C07272=1095.024,419.348,-100.142,178.825,23.629,153.449
C07273=1095.018,419.101,-100.102,178.823,23.620,153.447
C07274=1095.011,418.855,-100.061,178.820,23.611,153.445
C07275=1095.006,418.608,-100.020,178.817,23.601,153.443
C07276=1095.000,418.362,-99.979,178.814,23.592,153.441
C07277=1094.993,418.116,-99.938,178.811,23.583,153.439
C07278=1094.987,417.868,-99.897,178.808,23.573,153.437
C07279=1094.982,417.653,-99.862,178.806,23.565,153.436
C07280=1094.976,417.437,-99.827,178.804,23.558,153.434
C07281=1094.972,417.222,-99.791,178.802,23.550,153.433
C07282=1094.966,417.006,-99.756,178.799,23.542,153.431
C07283=1094.960,416.791,-99.720,178.797,23.534,153.429
C07284=1094.956,416.575,-99.685,178.794,23.526,153.428
C07285=1094.950,416.359,-99.649,178.792,23.518,153.426
C07286=1094.945,416.144,-99.613,178.789,23.510,153.424
C07287=1094.938,415.897,-99.573,178.786,23.501,153.423
C07288=1094.933,415.650,-99.533,178.783,23.492,153.421
C07289=1094.926,415.404,-99.492,178.780,23.483,153.419
C07290=1094.920,415.157,-99.452,178.778,23.475,153.417
C07291=1094.914,414.910,-99.411,178.776,23.466,153.415
C07292=1094.908,414.664,-99.371,178.772,23.457,153.414
C07293=1094.902,414.417,-99.331,178.770,23.448,153.412
C07294=1094.896,414.170,-99.290,178.767,23.439,153.410
C07295=1094.890,413.923,-99.251,178.764,23.431,153.408
C07296=1094.883,413.677,-99.211,178.762,23.422,153.407
C07297=1094.877,413.430,-99.171,178.758,23.414,153.405
C07298=1094.871,413.184,-99.130,178.756,23.405,153.403
C07299=1094.865,412.937,-99.090,178.753,23.396,153.401
C07300=1094.859,412.690,-99.050,178.750,23.387,153.400
C07301=1094.853,412.443,-99.010,178.747,23.379,153.398
C07302=1094.847,412.197,-98.970,178.744,23.371,153.396
C07303=1094.841,411.951,-98.930,178.741,23.362,153.395
C07304=1094.835,411.704,-98.890,178.738,23.353,153.393
C07305=1094.829,411.457,-98.850,178.736,23.345,153.391
C07306=1094.823,411.210,-98.809,178.733,23.337,153.390
C07307=1094.816,410.955,-98.768,178.730,23.328,153.388
C07308=1094.810,410.698,-98.727,178.727,23.319,153.386
C07309=1094.804,410.442,-98.686,178.724,23.311,153.384
C07310=1094.798,410.186,-98.644,178.721,23.302,153.383
C07311=1094.791,409.939,-98.604,178.719,23.294,153.381
C07312=1094.785,409.692,-98.565,178.716,23.286,153.379
C07313=1094.780,409.446,-98.524,178.713,23.277,153.378
C07314=1094.774,409.199,-98.485,178.711,23.269,153.376
C07315=1094.768,408.952,-98.445,178.708,23.261,153.374
C07316=1094.762,408.705,-98.405,178.705,23.253,153.373
C07317=1094.755,408.459,-98.365,178.702,23.245,153.371
C07318=1094.750,408.212,-98.326,178.699,23.237,153.370
C07319=1094.744,407.965,-98.287,178.696,23.228,153.368
C07320=1094.738,407.718,-98.246,178.694,23.220,153.366
C07321=1094.732,407.471,-98.207,178.691,23.212,153.365
C07322=1094.727,407.225,-98.167,178.688,23.205,153.363
C07323=1094.720,406.978,-98.127,178.685,23.196,153.362
C07324=1094.714,406.731,-98.088,178.682,23.188,153.360
C07325=1094.708,406.484,-98.048,178.680,23.180,153.359
C07326=1094.703,406.237,-98.009,178.677,23.172,153.357
C07327=1094.695,405.991,-97.970,178.674,23.164,153.356
C07328=1094.689,405.744,-97.930,178.671,23.156,153.354
C07329=1094.683,405.497,-97.891,178.669,23.149,153.353
C07330=1094.678,405.250,-97.852,178.666,23.141,153.351
C07331=1094.672,405.003,-97.812,178.663,23.133,153.349
C07332=1094.666,404.756,-97.773,178.660,23.126,153.348
C07333=1094.660,404.510,-97.734,178.657,23.118,153.347
C07334=1094.654,404.263,-97.695,178.655,23.110,153.345
C07335=1094.648,404.015,-97.655,178.651,23.102,153.344
C07336=1094.642,403.769,-97.617,178.649,23.095,153.342
C07337=1094.636,403.522,-97.577,178.646,23.087,153.341
C07338=1094.630,403.275,-97.538,178.643,23.080,153.339
C07339=1094.624,403.029,-97.499,178.640,23.072,153.338
C07340=1094.617,402.782,-97.460,178.638,23.064,153.336
C07341=1094.611,402.535,-97.420,178.635,23.057,153.335
C07342=1094.606,402.288,-97.381,178.632,23.049,153.333
C07343=1094.600,402.041,-97.342,178.630,23.042,153.332
C07344=1094.593,401.794,-97.303,178.626,23.034,153.331
C07345=1094.588,401.548,-97.264,178.624,23.027,153.329
C07346=1094.581,401.301,-97.225,178.620,23.019,153.328
C07347=1094.576,401.054,-97.186,178.618,23.012,153.326
C07348=1094.569,400.807,-97.147,178.615,23.005,153.325
C07349=1094.564,400.560,-97.108,178.612,22.997,153.324
C07350=1094.558,400.313,-97.069,178.610,22.990,153.322
C07351=1094.551,400.066,-97.031,178.607,22.982,153.321
C07352=1094.546,399.819,-96.992,178.604,22.975,153.319
C07353=1094.540,399.572,-96.952,178.601,22.968,153.318
C07354=1094.534,399.326,-96.915,178.598,22.961,153.317
C07355=1094.528,399.078,-96.875,178.596,22.954,153.315
C07356=1094.522,398.832,-96.837,178.592,22.946,153.314
C07357=1094.516,398.584,-96.798,178.590,22.939,153.313
C07358=1094.510,398.338,-96.759,178.587,22.932,153.311
C07359=1094.504,398.118,-96.725,178.585,22.926,153.310
C07360=1094.499,397.898,-96.691,178.582,22.919,153.309
C07361=1094.493,397.677,-96.656,178.579,22.913,153.308
C07362=1094.489,397.458,-96.621,178.577,22.907,153.306
C07363=1094.483,397.237,-96.586,178.575,22.900,153.305
C07364=1094.478,397.017,-96.552,178.572,22.894,153.304
C07365=1094.473,396.798,-96.518,178.569,22.888,153.303
C07366=1094.468,396.577,-96.484,178.567,22.882,153.302
C07367=1094.461,396.331,-96.445,178.564,22.874,153.301
C07368=1094.455,396.083,-96.407,178.561,22.868,153.299
C07369=1094.450,395.836,-96.369,178.559,22.861,153.298
C07370=1094.443,395.590,-96.330,178.556,22.854,153.297
C07371=1094.438,395.343,-96.292,178.553,22.847,153.295
C07372=1094.432,395.096,-96.254,178.550,22.840,153.294
C07373=1094.426,394.849,-96.214,178.548,22.833,153.293
C07374=1094.420,394.602,-96.177,178.544,22.826,153.292
C07375=1094.414,394.355,-96.139,178.541,22.819,153.290
C07376=1094.408,394.108,-96.099,178.539,22.813,153.289
C07377=1094.402,393.861,-96.062,178.536,22.806,153.288
C07378=1094.396,393.615,-96.024,178.533,22.799,153.287
C07379=1094.390,393.367,-95.985,178.530,22.792,153.285
C07380=1094.384,393.121,-95.947,178.527,22.786,153.284
C07381=1094.378,392.874,-95.909,178.525,22.779,153.283
C07382=1094.372,392.626,-95.871,178.521,22.772,153.282
C07383=1094.366,392.379,-95.833,178.519,22.765,153.281
C07384=1094.361,392.133,-95.795,178.516,22.759,153.279
C07385=1094.354,391.885,-95.757,178.513,22.752,153.278
C07386=1094.348,391.638,-95.719,178.511,22.746,153.277
C07387=1094.342,391.392,-95.681,178.507,22.739,153.276
C07388=1094.336,391.144,-95.643,178.504,22.732,153.275
C07389=1094.330,390.898,-95.605,178.502,22.726,153.274
C07390=1094.324,390.651,-95.566,178.499,22.720,153.272
C07391=1094.318,390.403,-95.529,178.496,22.713,153.271
C07392=1094.312,390.156,-95.491,178.493,22.706,153.270
C07393=1094.306,389.910,-95.453,178.490,22.700,153.269
C07394=1094.300,389.663,-95.416,178.487,22.694,153.268
C07395=1094.295,389.416,-95.378,178.485,22.687,153.267
C07396=1094.288,389.169,-95.340,178.482,22.681,153.266
C07397=1094.282,388.922,-95.302,178.478,22.674,153.265
C07398=1094.276,388.675,-95.264,178.475,22.668,153.263
C07399=1094.270,388.428,-95.226,178.473,22.662,153.262
C07400=1094.264,388.182,-95.189,178.470,22.655,153.261
C07401=1094.258,387.934,-95.151,178.467,22.649,153.260
C07402=1094.252,387.687,-95.113,178.464,22.643,153.259
C07403=1094.246,387.440,-95.076,178.461,22.636,153.258
C07404=1094.240,387.193,-95.038,178.458,22.630,153.257
C07405=1094.235,386.947,-95.000,178.455,22.624,153.256
C07406=1094.229,386.699,-94.963,178.452,22.617,153.254
C07407=1094.223,386.453,-94.925,178.450,22.611,153.253
C07408=1094.217,386.205,-94.887,178.447,22.605,153.252
C07409=1094.211,385.958,-94.850,178.444,22.599,153.251
C07410=1094.205,385.711,-94.812,178.441,22.593,153.250
C07411=1094.199,385.464,-94.775,178.438,22.586,153.249
C07412=1094.194,385.217,-94.738,178.435,22.580,153.248
C07413=1094.188,384.970,-94.700,178.432,22.574,153.247
C07414=1094.182,384.723,-94.663,178.429,22.568,153.246
C07415=1094.177,384.509,-94.630,178.427,22.563,153.245
C07416=1094.172,384.296,-94.598,178.424,22.557,153.244
C07417=1094.166,384.082,-94.566,178.422,22.552,153.243
C07418=1094.161,383.869,-94.534,178.420,22.547,153.242
C07419=1094.156,383.655,-94.502,178.417,22.542,153.242
C07420=1094.151,383.441,-94.469,178.415,22.536,153.240
C07421=1094.146,383.228,-94.437,178.411,22.531,153.240
C07422=1094.142,383.014,-94.405,178.409,22.525,153.239
C07423=1094.136,382.767,-94.367,178.406,22.519,153.238
C07424=1094.130,382.520,-94.330,178.404,22.514,153.237
C07425=1094.124,382.273,-94.294,178.401,22.508,153.236
C07426=1094.118,382.026,-94.256,178.398,22.502,153.235
C07427=1094.112,381.778,-94.218,178.395,22.496,153.234
C07428=1094.105,381.531,-94.182,178.392,22.490,153.233
C07429=1094.099,381.284,-94.144,178.389,22.485,153.232
C07430=1094.094,381.037,-94.107,178.386,22.479,153.231
C07431=1094.087,380.790,-94.071,178.383,22.473,153.230
C07432=1094.081,380.543,-94.033,178.380,22.467,153.229
C07433=1094.076,380.296,-93.996,178.377,22.461,153.228
C07434=1094.070,380.049,-93.959,178.374,22.455,153.227
C07435=1094.064,379.801,-93.922,178.371,22.450,153.226
C07436=1094.058,379.554,-93.885,178.369,22.444,153.225
C07437=1094.052,379.308,-93.849,178.366,22.438,153.224
C07438=1094.047,379.061,-93.812,178.363,22.432,153.223
C07439=1094.040,378.814,-93.775,178.360,22.427,153.222
C07440=1094.035,378.567,-93.738,178.357,22.421,153.221
C07441=1094.029,378.319,-93.701,178.354,22.415,153.220
C07442=1094.023,378.072,-93.665,178.351,22.409,153.220
C07443=1094.017,377.825,-93.628,178.348,22.403,153.218
C07444=1094.011,377.578,-93.591,178.345,22.398,153.218
C07445=1094.005,377.330,-93.554,178.342,22.392,153.217
C07446=1093.999,377.083,-93.518,178.339,22.386,153.216
C07447=1093.993,376.836,-93.481,178.336,22.381,153.215
C07448=1093.988,376.589,-93.444,178.333,22.375,153.214
C07449=1093.982,376.342,-93.407,178.330,22.370,153.213
C07450=1093.976,376.095,-93.370,178.327,22.364,153.212
C07451=1093.970,375.848,-93.334,178.324,22.358,153.211
C07452=1093.965,375.600,-93.297,178.321,22.353,153.210
C07453=1093.958,375.353,-93.261,178.318,22.347,153.209
C07454=1093.953,375.105,-93.224,178.315,22.342,153.209
C07455=1093.947,374.859,-93.188,178.312,22.336,153.208
C07456=1093.942,374.612,-93.151,178.309,22.331,153.207
C07457=1093.935,374.365,-93.115,178.307,22.325,153.206
C07458=1093.930,374.117,-93.078,178.304,22.320,153.205
C07459=1093.924,373.870,-93.042,178.301,22.314,153.204
C07460=1093.917,373.623,-93.005,178.298,22.309,153.203
C07461=1093.912,373.376,-92.969,178.295,22.304,153.203
C07462=1093.906,373.129,-92.932,178.292,22.298,153.202
C07463=1093.900,372.881,-92.897,178.289,22.293,153.201
C07464=1093.894,372.634,-92.860,178.285,22.287,153.200
C07465=1093.888,372.387,-92.823,178.282,22.282,153.199
C07466=1093.883,372.140,-92.788,178.280,22.277,153.198
C07467=1093.876,371.893,-92.751,178.277,22.272,153.198
C07468=1093.871,371.645,-92.715,178.274,22.266,153.197
C07469=1093.865,371.398,-92.678,178.271,22.261,153.196
C07470=1093.858,371.151,-92.642,178.268,22.255,153.195
C07471=1093.849,370.751,-92.584,178.263,22.247,153.194
C07472=1093.840,370.351,-92.526,178.258,22.238,153.192
C07473=1093.830,369.951,-92.467,178.254,22.230,153.191
C07474=1093.821,369.552,-92.409,178.249,22.222,153.190
C07475=1093.815,369.304,-92.373,178.246,22.217,153.189
C07476=1093.808,369.057,-92.337,178.243,22.211,153.188
C07477=1093.804,368.810,-92.301,178.240,22.206,153.187
C07478=1093.798,368.562,-92.265,178.236,22.201,153.187
C07479=1093.791,368.315,-92.229,178.234,22.196,153.186
C07480=1093.785,368.067,-92.193,178.231,22.190,153.185
C07481=1093.780,367.820,-92.157,178.228,22.185,153.184
C07482=1093.774,367.573,-92.120,178.225,22.180,153.184
C07483=1093.769,367.326,-92.085,178.222,22.175,153.183
C07484=1093.763,367.078,-92.049,178.218,22.170,153.182
C07485=1093.757,366.831,-92.014,178.216,22.165,153.181
C07486=1093.751,366.584,-91.977,178.213,22.160,153.180
C07487=1093.745,366.337,-91.942,178.210,22.155,153.180
C07488=1093.739,366.089,-91.906,178.207,22.150,153.179
C07489=1093.734,365.842,-91.871,178.204,22.144,153.178
C07490=1093.728,365.594,-91.835,178.201,22.140,153.177
C07491=1093.722,365.347,-91.799,178.198,22.135,153.177
C07492=1093.716,365.100,-91.763,178.195,22.130,153.176
C07493=1093.710,364.853,-91.727,178.192,22.125,153.175
C07494=1093.704,364.606,-91.692,178.189,22.120,153.175
C07495=1093.698,364.358,-91.656,178.186,22.115,153.174
C07496=1093.692,364.110,-91.621,178.183,22.110,153.173
C07497=1093.687,363.863,-91.585,178.180,22.105,153.172
C07498=1093.681,363.616,-91.549,178.177,22.101,153.172
C07499=1093.675,363.369,-91.514,178.174,22.095,153.171
C07500=1093.669,363.121,-91.478,178.171,22.090,153.170
C07501=1093.663,362.873,-91.443,178.168,22.085,153.170
C07502=1093.658,362.626,-91.407,178.165,22.081,153.169
C07503=1093.652,362.379,-91.372,178.162,22.076,153.168
C07504=1093.647,362.132,-91.336,178.159,22.071,153.168
C07505=1093.640,361.884,-91.301,178.156,22.066,153.167
C07506=1093.635,361.637,-91.266,178.153,22.061,153.166
C07507=1093.629,361.389,-91.231,178.150,22.057,153.166
C07508=1093.623,361.141,-91.195,178.147,22.052,153.165
C07509=1093.617,360.894,-91.160,178.143,22.047,153.164
C07510=1093.611,360.647,-91.124,178.141,22.042,153.163
C07511=1093.605,360.400,-91.089,178.138,22.038,153.163
C07512=1093.599,360.152,-91.054,178.135,22.032,153.162
C07513=1093.594,359.905,-91.019,178.132,22.028,153.161
C07514=1093.588,359.657,-90.983,178.129,22.024,153.161
C07515=1093.583,359.409,-90.948,178.126,22.018,153.160
C07516=1093.576,359.162,-90.913,178.122,22.014,153.160
C07517=1093.570,358.915,-90.878,178.120,22.009,153.159
C07518=1093.564,358.667,-90.842,178.117,22.004,153.158
C07519=1093.559,358.420,-90.808,178.113,22.000,153.158
C07520=1093.553,358.172,-90.772,178.111,21.995,153.157
C07521=1093.547,357.925,-90.738,178.107,21.991,153.156
C07522=1093.541,357.678,-90.703,178.104,21.986,153.156
C07523=1093.532,357.293,-90.649,178.100,21.979,153.155
C07524=1093.523,356.908,-90.593,178.095,21.972,153.154
C07525=1093.514,356.524,-90.539,178.091,21.965,153.153
C07526=1093.505,356.139,-90.485,178.085,21.957,153.152
C07527=1093.499,355.892,-90.450,178.083,21.953,153.151
C07528=1093.493,355.644,-90.415,178.080,21.948,153.151
C07529=1093.488,355.397,-90.380,178.076,21.943,153.150
C07530=1093.482,355.150,-90.346,178.074,21.939,153.149
C07531=1093.476,354.902,-90.310,178.070,21.934,153.149
C07532=1093.470,354.655,-90.276,178.067,21.930,153.148
C07533=1093.464,354.406,-90.241,178.065,21.926,153.147
C07534=1093.459,354.160,-90.206,178.061,21.921,153.147
C07535=1093.453,353.912,-90.172,178.059,21.917,153.146
C07536=1093.447,353.664,-90.137,178.055,21.912,153.146
C07537=1093.441,353.417,-90.102,178.052,21.908,153.145
C07538=1093.436,353.170,-90.067,178.049,21.903,153.145
C07539=1093.430,352.922,-90.033,178.046,21.899,153.144
C07540=1093.425,352.674,-89.998,178.043,21.894,153.143
C07541=1093.418,352.427,-89.963,178.040,21.890,153.143
C07542=1093.412,352.179,-89.929,178.037,21.886,153.142
C07543=1093.407,351.932,-89.894,178.034,21.881,153.142
C07544=1093.400,351.684,-89.860,178.031,21.877,153.141
C07545=1093.395,351.436,-89.825,178.027,21.872,153.141
C07546=1093.389,351.190,-89.791,178.025,21.868,153.140
C07547=1093.383,350.942,-89.756,178.021,21.864,153.140
C07548=1093.377,350.694,-89.721,178.019,21.860,153.139
C07549=1093.372,350.447,-89.687,178.016,21.855,153.138
C07550=1093.367,350.199,-89.653,178.012,21.851,153.138
C07551=1093.360,349.951,-89.618,178.010,21.846,153.137
C07552=1093.354,349.704,-89.584,178.006,21.842,153.137
C07553=1093.349,349.456,-89.550,178.004,21.838,153.136
C07554=1093.343,349.208,-89.515,178.000,21.834,153.136
C07555=1093.337,348.961,-89.481,177.998,21.829,153.135
C07556=1093.332,348.713,-89.447,177.994,21.825,153.135
C07557=1093.326,348.466,-89.412,177.992,21.821,153.134
C07558=1093.319,348.218,-89.378,177.988,21.817,153.134
C07559=1093.313,347.971,-89.344,177.985,21.812,153.133
C07560=1093.308,347.723,-89.309,177.982,21.808,153.133
C07561=1093.302,347.476,-89.275,177.979,21.804,153.132
C07562=1093.296,347.228,-89.241,177.976,21.800,153.131
C07563=1093.291,346.980,-89.206,177.973,21.795,153.131
C07564=1093.285,346.733,-89.173,177.970,21.791,153.130
C07565=1093.279,346.485,-89.139,177.967,21.787,153.130
C07566=1093.274,346.238,-89.105,177.964,21.783,153.129
C07567=1093.268,345.991,-89.071,177.961,21.778,153.129
C07568=1093.262,345.742,-89.036,177.958,21.775,153.128
C07569=1093.256,345.494,-89.002,177.955,21.770,153.128
C07570=1093.251,345.247,-88.968,177.951,21.766,153.127
C07571=1093.245,345.000,-88.934,177.949,21.762,153.127
C07572=1093.239,344.753,-88.900,177.945,21.758,153.126
C07573=1093.233,344.504,-88.866,177.942,21.754,153.126
C07574=1093.228,344.256,-88.832,177.939,21.750,153.125
C07575=1093.219,343.874,-88.780,177.934,21.743,153.125
C07576=1093.209,343.492,-88.727,177.930,21.737,153.124
C07577=1093.201,343.110,-88.676,177.925,21.731,153.123
C07578=1093.191,342.728,-88.623,177.921,21.725,153.123
C07579=1093.186,342.481,-88.589,177.917,21.721,153.122
C07580=1093.180,342.233,-88.555,177.914,21.717,153.122
C07581=1093.174,341.985,-88.522,177.911,21.713,153.121
C07582=1093.168,341.738,-88.488,177.908,21.709,153.121
C07583=1093.163,341.490,-88.455,177.905,21.705,153.120
C07584=1093.157,341.243,-88.421,177.902,21.701,153.120
C07585=1093.151,340.995,-88.387,177.899,21.697,153.119
C07586=1093.146,340.748,-88.353,177.896,21.693,153.119
C07587=1093.140,340.500,-88.320,177.892,21.688,153.118
C07588=1093.134,340.252,-88.285,177.890,21.685,153.118
C07589=1093.128,340.004,-88.252,177.886,21.680,153.117
C07590=1093.122,339.756,-88.219,177.883,21.677,153.117
C07591=1093.117,339.509,-88.185,177.881,21.673,153.117
C07592=1093.111,339.261,-88.151,177.877,21.669,153.116
C07593=1093.106,339.013,-88.118,177.875,21.665,153.116
C07594=1093.100,338.766,-88.084,177.871,21.661,153.115
C07595=1093.094,338.518,-88.051,177.868,21.657,153.115
C07596=1093.088,338.270,-88.018,177.865,21.653,153.114
C07597=1093.082,338.023,-87.984,177.862,21.650,153.114
C07598=1093.076,337.775,-87.950,177.859,21.646,153.113
C07599=1093.071,337.527,-87.917,177.856,21.642,153.113
C07600=1093.065,337.279,-87.884,177.853,21.638,153.113
C07601=1093.059,337.032,-87.851,177.850,21.634,153.112
C07602=1093.053,336.784,-87.817,177.847,21.630,153.112
C07603=1093.048,336.536,-87.784,177.843,21.626,153.111
C07604=1093.042,336.288,-87.750,177.840,21.623,153.111
C07605=1093.036,336.041,-87.718,177.838,21.619,153.111
C07606=1093.030,335.793,-87.684,177.834,21.615,153.110
C07607=1093.025,335.545,-87.651,177.831,21.611,153.110
C07608=1093.019,335.298,-87.617,177.828,21.607,153.109
C07609=1093.012,335.050,-87.584,177.825,21.604,153.109
C07610=1093.007,334.802,-87.551,177.822,21.600,153.109
C07611=1093.001,334.554,-87.517,177.819,21.596,153.108
C07612=1092.996,334.306,-87.484,177.816,21.592,153.108
C07613=1092.989,334.059,-87.451,177.812,21.589,153.107
C07614=1092.984,333.811,-87.418,177.810,21.585,153.107
C07615=1092.979,333.564,-87.385,177.807,21.581,153.107
C07616=1092.973,333.316,-87.352,177.803,21.577,153.106
C07617=1092.967,333.068,-87.319,177.801,21.574,153.106
C07618=1092.962,332.820,-87.286,177.798,21.570,153.105
C07619=1092.955,332.573,-87.253,177.794,21.566,153.105
C07620=1092.950,332.324,-87.220,177.792,21.562,153.105
C07621=1092.944,332.076,-87.187,177.788,21.559,153.104
C07622=1092.938,331.829,-87.154,177.785,21.555,153.104
C07623=1092.933,331.581,-87.121,177.782,21.551,153.103
C07624=1092.926,331.333,-87.088,177.779,21.548,153.103
C07625=1092.920,331.086,-87.055,177.776,21.544,153.103
C07626=1092.915,330.838,-87.022,177.773,21.541,153.103
C07627=1092.905,330.450,-86.971,177.768,21.535,153.102
C07628=1092.896,330.062,-86.920,177.763,21.529,153.101
C07629=1092.887,329.674,-86.868,177.758,21.524,153.101
C07630=1092.878,329.286,-86.817,177.754,21.518,153.100
C07631=1092.872,329.039,-86.785,177.750,21.515,153.100
C07632=1092.867,328.790,-86.752,177.747,21.511,153.100
C07633=1092.861,328.542,-86.719,177.745,21.508,153.099
C07634=1092.854,328.295,-86.686,177.741,21.504,153.099
C07635=1092.849,328.046,-86.654,177.738,21.501,153.099
C07636=1092.843,327.799,-86.621,177.735,21.497,153.098
C07637=1092.837,327.551,-86.589,177.732,21.493,153.098
C07638=1092.832,327.303,-86.556,177.729,21.490,153.098
C07639=1092.826,327.056,-86.523,177.726,21.487,153.097
C07640=1092.820,326.808,-86.491,177.722,21.482,153.097
C07641=1092.815,326.560,-86.458,177.720,21.479,153.097
C07642=1092.809,326.312,-86.426,177.717,21.476,153.096
C07643=1092.802,326.065,-86.394,177.714,21.472,153.096
C07644=1092.797,325.816,-86.361,177.710,21.469,153.096
C07645=1092.791,325.569,-86.329,177.707,21.465,153.095
C07646=1092.785,325.321,-86.297,177.705,21.462,153.095
C07647=1092.780,325.073,-86.263,177.701,21.458,153.095
C07648=1092.774,324.825,-86.231,177.698,21.455,153.094
C07649=1092.768,324.578,-86.199,177.695,21.452,153.094
C07650=1092.762,324.330,-86.167,177.692,21.448,153.094
C07651=1092.757,324.081,-86.134,177.688,21.445,153.093
C07652=1092.751,323.834,-86.101,177.686,21.441,153.093
C07653=1092.745,323.586,-86.070,177.683,21.438,153.093
C07654=1092.739,323.338,-86.037,177.680,21.435,153.092
C07655=1092.734,323.090,-86.004,177.676,21.431,153.092
C07656=1092.728,322.842,-85.973,177.673,21.427,153.092
C07657=1092.722,322.594,-85.941,177.671,21.424,153.091
C07658=1092.716,322.347,-85.908,177.668,21.421,153.091
C07659=1092.711,322.099,-85.876,177.664,21.417,153.091
C07660=1092.705,321.851,-85.844,177.661,21.414,153.091
C07661=1092.700,321.604,-85.811,177.658,21.410,153.090
C07662=1092.694,321.355,-85.779,177.655,21.407,153.090
C07663=1092.688,321.107,-85.747,177.652,21.403,153.090
C07664=1092.682,320.860,-85.716,177.649,21.400,153.089
C07665=1092.677,320.611,-85.683,177.646,21.397,153.089
C07666=1092.671,320.364,-85.650,177.643,21.394,153.089
C07667=1092.665,320.116,-85.619,177.639,21.390,153.089
C07668=1092.659,319.868,-85.587,177.637,21.386,153.088
C07669=1092.654,319.620,-85.555,177.634,21.383,153.088
C07670=1092.648,319.372,-85.523,177.631,21.380,153.088
C07671=1092.643,319.124,-85.491,177.627,21.376,153.087
C07672=1092.637,318.876,-85.459,177.624,21.373,153.087
C07673=1092.632,318.629,-85.427,177.621,21.370,153.087
C07674=1092.626,318.380,-85.395,177.619,21.366,153.086
C07675=1092.621,318.133,-85.363,177.616,21.363,153.086
C07676=1092.615,317.885,-85.331,177.612,21.360,153.086
C07677=1092.609,317.637,-85.300,177.609,21.356,153.086
C07678=1092.603,317.389,-85.267,177.606,21.353,153.085
C07679=1092.595,316.994,-85.216,177.601,21.347,153.085
C07680=1092.586,316.599,-85.165,177.597,21.343,153.084
C07681=1092.577,316.204,-85.115,177.592,21.337,153.084
C07682=1092.568,315.809,-85.065,177.587,21.332,153.083
C07683=1092.563,315.562,-85.032,177.584,21.328,153.083
C07684=1092.557,315.313,-85.000,177.581,21.325,153.083
C07685=1092.552,315.066,-84.969,177.578,21.322,153.083
C07686=1092.545,314.818,-84.937,177.574,21.319,153.082
C07687=1092.540,314.570,-84.906,177.571,21.315,153.082
C07688=1092.534,314.322,-84.874,177.568,21.312,153.082
C07689=1092.527,314.074,-84.843,177.565,21.309,153.082
C07690=1092.522,313.826,-84.811,177.562,21.306,153.081
C07691=1092.516,313.578,-84.779,177.559,21.303,153.081
C07692=1092.511,313.330,-84.748,177.556,21.299,153.081
C07693=1092.504,313.082,-84.717,177.553,21.296,153.081
C07694=1092.499,312.834,-84.685,177.550,21.293,153.081
C07695=1092.493,312.586,-84.653,177.547,21.290,153.080
C07696=1092.487,312.338,-84.623,177.544,21.287,153.080
C07697=1092.481,312.091,-84.591,177.541,21.284,153.080
C07698=1092.475,311.843,-84.559,177.537,21.281,153.080
C07699=1092.470,311.595,-84.529,177.534,21.277,153.079
C07700=1092.464,311.347,-84.497,177.531,21.275,153.079
C07701=1092.458,311.099,-84.466,177.528,21.272,153.079
C07702=1092.452,310.851,-84.434,177.525,21.268,153.079
C07703=1092.446,310.603,-84.403,177.522,21.265,153.078
C07704=1092.441,310.355,-84.372,177.519,21.262,153.078
C07705=1092.435,310.107,-84.340,177.515,21.259,153.078
C07706=1092.429,309.859,-84.309,177.513,21.256,153.078
C07707=1092.423,309.611,-84.278,177.509,21.253,153.078
C07708=1092.418,309.363,-84.247,177.506,21.250,153.077
C07709=1092.412,309.115,-84.215,177.503,21.247,153.077
C07710=1092.406,308.867,-84.185,177.501,21.244,153.077
C07711=1092.400,308.619,-84.153,177.498,21.241,153.077
C07712=1092.395,308.372,-84.123,177.494,21.237,153.077
C07713=1092.389,308.123,-84.091,177.491,21.234,153.076
C07714=1092.383,307.875,-84.060,177.488,21.231,153.076
C07715=1092.377,307.628,-84.028,177.485,21.228,153.076
C07716=1092.372,307.379,-83.997,177.482,21.225,153.076
C07717=1092.366,307.132,-83.966,177.479,21.222,153.075
C07718=1092.361,306.884,-83.935,177.476,21.219,153.075
C07719=1092.354,306.635,-83.904,177.472,21.216,153.075
C07720=1092.349,306.388,-83.873,177.469,21.213,153.075
C07721=1092.343,306.140,-83.842,177.466,21.210,153.075
C07722=1092.338,305.892,-83.811,177.463,21.207,153.074
C07723=1092.331,305.644,-83.780,177.460,21.204,153.074
C07724=1092.326,305.396,-83.749,177.457,21.201,153.074
C07725=1092.320,305.148,-83.719,177.454,21.198,153.074
C07726=1092.315,304.900,-83.688,177.451,21.195,153.074
C07727=1092.309,304.653,-83.657,177.447,21.191,153.073
C07728=1092.303,304.404,-83.625,177.444,21.188,153.073
C07729=1092.298,304.156,-83.595,177.441,21.185,153.073
C07730=1092.292,303.908,-83.564,177.438,21.183,153.073
C07731=1092.283,303.516,-83.515,177.434,21.178,153.072
C07732=1092.274,303.123,-83.467,177.429,21.173,153.072
C07733=1092.265,302.732,-83.418,177.424,21.168,153.072
C07734=1092.257,302.339,-83.369,177.419,21.163,153.072
C07735=1092.251,302.091,-83.339,177.416,21.160,153.071
C07736=1092.246,301.843,-83.308,177.413,21.157,153.071
C07737=1092.240,301.595,-83.277,177.410,21.154,153.071
C07738=1092.234,301.347,-83.247,177.407,21.151,153.071
C07739=1092.229,301.099,-83.216,177.404,21.149,153.071
C07740=1092.223,300.851,-83.186,177.401,21.146,153.070
C07741=1092.218,300.603,-83.155,177.398,21.143,153.070
C07742=1092.212,300.355,-83.124,177.395,21.140,153.070
C07743=1092.206,300.107,-83.094,177.391,21.136,153.070
C07744=1092.201,299.858,-83.063,177.388,21.133,153.070
C07745=1092.195,299.611,-83.032,177.385,21.130,153.069
C07746=1092.189,299.363,-83.002,177.382,21.127,153.069
C07747=1092.184,299.115,-82.971,177.379,21.124,153.069
C07748=1092.178,298.867,-82.941,177.376,21.121,153.069
C07749=1092.173,298.619,-82.910,177.373,21.118,153.069
C07750=1092.167,298.371,-82.879,177.370,21.115,153.068
C07751=1092.161,298.123,-82.849,177.367,21.113,153.068
C07752=1092.156,297.875,-82.819,177.364,21.110,153.068
C07753=1092.151,297.627,-82.789,177.361,21.107,153.068
C07754=1092.145,297.379,-82.758,177.358,21.104,153.068
C07755=1092.139,297.131,-82.728,177.355,21.101,153.068
C07756=1092.133,296.883,-82.697,177.352,21.098,153.068
C07757=1092.127,296.634,-82.667,177.349,21.096,153.067
C07758=1092.121,296.386,-82.637,177.346,21.093,153.067
C07759=1092.116,296.138,-82.607,177.343,21.090,153.067
C07760=1092.111,295.890,-82.576,177.340,21.087,153.067
C07761=1092.105,295.642,-82.546,177.337,21.084,153.067
C07762=1092.099,295.394,-82.516,177.334,21.081,153.067
C07763=1092.093,295.146,-82.485,177.331,21.078,153.066
C07764=1092.088,294.898,-82.456,177.328,21.076,153.066
C07765=1092.082,294.650,-82.425,177.325,21.073,153.066
C07766=1092.076,294.402,-82.395,177.321,21.070,153.066
C07767=1092.071,294.154,-82.366,177.318,21.067,153.066
C07768=1092.065,293.906,-82.335,177.315,21.064,153.066
C07769=1092.059,293.658,-82.305,177.312,21.061,153.065
C07770=1092.054,293.409,-82.275,177.309,21.058,153.065
C07771=1092.048,293.162,-82.245,177.305,21.056,153.065
C07772=1092.042,292.913,-82.215,177.302,21.053,153.065
C07773=1092.036,292.665,-82.185,177.299,21.050,153.065
C07774=1092.031,292.417,-82.155,177.296,21.047,153.065
C07775=1092.025,292.169,-82.125,177.293,21.044,153.065
C07776=1092.020,291.921,-82.095,177.290,21.041,153.065
C07777=1092.014,291.673,-82.065,177.287,21.038,153.064
C07778=1092.008,291.424,-82.035,177.284,21.036,153.064
C07779=1092.003,291.177,-82.005,177.281,21.033,153.064
C07780=1091.997,290.928,-81.975,177.278,21.030,153.064
C07781=1091.991,290.680,-81.946,177.275,21.027,153.064
C07782=1091.985,290.432,-81.916,177.272,21.025,153.064
C07783=1091.977,290.054,-81.870,177.267,21.020,153.063
C07784=1091.969,289.675,-81.825,177.262,21.016,153.063
C07785=1091.960,289.297,-81.779,177.258,21.012,153.063
C07786=1091.951,288.919,-81.734,177.253,21.008,153.063
C07787=1091.945,288.671,-81.705,177.250,21.005,153.063
C07788=1091.939,288.423,-81.675,177.247,21.003,153.063
C07789=1091.934,288.175,-81.645,177.244,21.000,153.063
C07790=1091.928,287.926,-81.615,177.241,20.997,153.062
C07791=1091.922,287.678,-81.586,177.238,20.994,153.062
C07792=1091.917,287.431,-81.556,177.235,20.992,153.062
C07793=1091.911,287.182,-81.527,177.232,20.989,153.062
C07794=1091.906,286.934,-81.497,177.229,20.986,153.062
C07795=1091.899,286.686,-81.468,177.226,20.984,153.062
C07796=1091.894,286.437,-81.438,177.223,20.981,153.062
C07797=1091.888,286.190,-81.408,177.220,20.979,153.062
C07798=1091.882,285.941,-81.379,177.217,20.976,153.061
C07799=1091.876,285.693,-81.349,177.214,20.973,153.061
C07800=1091.871,285.445,-81.320,177.211,20.970,153.061
C07801=1091.866,285.197,-81.290,177.208,20.968,153.061
C07802=1091.860,284.949,-81.261,177.204,20.965,153.061
C07803=1091.854,284.700,-81.232,177.202,20.962,153.061
C07804=1091.849,284.452,-81.202,177.198,20.960,153.061
C07805=1091.842,284.204,-81.173,177.195,20.957,153.061
C07806=1091.837,283.956,-81.144,177.192,20.954,153.061
C07807=1091.832,283.707,-81.114,177.189,20.951,153.060
C07808=1091.826,283.459,-81.085,177.186,20.948,153.060
C07809=1091.820,283.211,-81.055,177.183,20.946,153.060
C07810=1091.815,282.963,-81.026,177.180,20.943,153.060
C07811=1091.809,282.715,-80.997,177.177,20.941,153.060
C07812=1091.803,282.467,-80.968,177.175,20.938,153.060
C07813=1091.798,282.218,-80.938,177.171,20.936,153.060
C07814=1091.792,281.971,-80.909,177.168,20.933,153.060
C07815=1091.787,281.722,-80.880,177.165,20.930,153.060
C07816=1091.780,281.474,-80.851,177.162,20.927,153.059
C07817=1091.775,281.226,-80.821,177.159,20.925,153.059
C07818=1091.770,280.978,-80.792,177.156,20.922,153.059
C07819=1091.764,280.729,-80.763,177.153,20.919,153.059
C07820=1091.758,280.481,-80.734,177.149,20.917,153.059
C07821=1091.752,280.233,-80.705,177.146,20.914,153.059
C07822=1091.747,279.985,-80.676,177.143,20.912,153.059
C07823=1091.741,279.737,-80.646,177.140,20.909,153.059
C07824=1091.735,279.488,-80.618,177.138,20.907,153.059
C07825=1091.730,279.240,-80.588,177.135,20.904,153.059
C07826=1091.724,278.992,-80.560,177.132,20.901,153.058
C07827=1091.719,278.744,-80.530,177.128,20.899,153.058
C07828=1091.713,278.495,-80.502,177.125,20.896,153.058
C07829=1091.707,278.246,-80.472,177.122,20.893,153.058
C07830=1091.701,277.999,-80.443,177.119,20.891,153.058
C07831=1091.696,277.750,-80.415,177.116,20.888,153.058
C07832=1091.690,277.502,-80.385,177.113,20.886,153.058
C07833=1091.684,277.254,-80.357,177.111,20.883,153.058
C07834=1091.679,277.005,-80.328,177.108,20.881,153.058
C07835=1091.670,276.637,-80.285,177.103,20.877,153.058
C07836=1091.662,276.268,-80.242,177.098,20.873,153.058
C07837=1091.654,275.899,-80.199,177.093,20.869,153.057
C07838=1091.646,275.530,-80.157,177.090,20.865,153.057
C07839=1091.639,275.282,-80.128,177.086,20.863,153.057
C07840=1091.634,275.034,-80.100,177.083,20.860,153.057
C07841=1091.628,274.786,-80.071,177.080,20.858,153.057
C07842=1091.623,274.537,-80.042,177.077,20.855,153.057
C07843=1091.617,274.289,-80.013,177.074,20.852,153.057
C07844=1091.611,274.040,-79.985,177.071,20.850,153.057
C07845=1091.606,273.793,-79.955,177.068,20.847,153.057
C07846=1091.600,273.544,-79.927,177.065,20.845,153.057
C07847=1091.594,273.296,-79.898,177.062,20.842,153.057
C07848=1091.589,273.048,-79.870,177.059,20.840,153.056
C07849=1091.583,272.799,-79.840,177.056,20.837,153.056
C07850=1091.578,272.551,-79.812,177.053,20.834,153.056
C07851=1091.572,272.302,-79.784,177.050,20.832,153.056
C07852=1091.566,272.054,-79.755,177.046,20.830,153.056
C07853=1091.560,271.806,-79.727,177.044,20.828,153.056
C07854=1091.554,271.558,-79.699,177.041,20.825,153.056
C07855=1091.549,271.310,-79.670,177.038,20.822,153.056
C07856=1091.543,271.061,-79.641,177.035,20.820,153.056
C07857=1091.538,270.813,-79.613,177.032,20.817,153.056
C07858=1091.532,270.564,-79.585,177.028,20.814,153.056
C07859=1091.527,270.317,-79.556,177.026,20.812,153.056
C07860=1091.521,270.068,-79.528,177.023,20.810,153.056
C07861=1091.515,269.820,-79.500,177.020,20.807,153.056
C07862=1091.510,269.571,-79.471,177.017,20.804,153.055
C07863=1091.504,269.323,-79.442,177.013,20.802,153.055
C07864=1091.498,269.075,-79.414,177.010,20.800,153.055
C07865=1091.492,268.826,-79.386,177.008,20.798,153.055
C07866=1091.487,268.578,-79.358,177.005,20.795,153.055
C07867=1091.481,268.329,-79.329,177.002,20.792,153.055
C07868=1091.476,268.081,-79.301,176.998,20.790,153.055
C07869=1091.470,267.832,-79.273,176.995,20.787,153.055
C07870=1091.464,267.585,-79.244,176.992,20.785,153.055
C07871=1091.458,267.336,-79.216,176.990,20.783,153.055
C07872=1091.453,267.088,-79.188,176.987,20.780,153.055
C07873=1091.447,266.839,-79.160,176.984,20.777,153.055
C07874=1091.442,266.591,-79.132,176.980,20.775,153.055
C07875=1091.436,266.343,-79.104,176.977,20.772,153.055
C07876=1091.430,266.095,-79.076,176.975,20.770,153.055
C07877=1091.425,265.847,-79.048,176.972,20.768,153.055
C07878=1091.419,265.598,-79.019,176.969,20.765,153.054
C07879=1091.414,265.350,-78.991,176.965,20.763,153.054
C07880=1091.408,265.101,-78.963,176.962,20.760,153.054
C07881=1091.403,264.853,-78.935,176.959,20.758,153.054
C07882=1091.397,264.604,-78.907,176.957,20.756,153.054
C07883=1091.391,264.356,-78.879,176.954,20.753,153.054
C07884=1091.385,264.108,-78.851,176.950,20.750,153.054
C07885=1091.380,263.859,-78.824,176.947,20.748,153.054
C07886=1091.374,263.611,-78.796,176.944,20.745,153.054
C07887=1091.365,263.245,-78.755,176.940,20.742,153.054
C07888=1091.356,262.879,-78.714,176.935,20.738,153.054
C07889=1091.348,262.512,-78.672,176.931,20.735,153.054
C07890=1091.340,262.146,-78.632,176.926,20.732,153.054
C07891=1091.333,261.898,-78.604,176.923,20.729,153.054
C07892=1091.328,261.650,-78.576,176.921,20.727,153.054
C07893=1091.322,261.401,-78.548,176.918,20.725,153.054
C07894=1091.316,261.153,-78.521,176.914,20.723,153.054
C07895=1091.311,260.905,-78.493,176.911,20.720,153.054
C07896=1091.305,260.656,-78.465,176.908,20.717,153.054
C07897=1091.299,260.408,-78.437,176.906,20.715,153.054
C07898=1091.293,260.159,-78.410,176.903,20.713,153.054
C07899=1091.288,259.911,-78.382,176.899,20.710,153.054
C07900=1091.282,259.663,-78.354,176.896,20.708,153.054
C07901=1091.276,259.414,-78.327,176.894,20.706,153.054
C07902=1091.271,259.166,-78.299,176.891,20.703,153.053
C07903=1091.265,258.918,-78.271,176.887,20.701,153.053
C07904=1091.259,258.669,-78.244,176.884,20.698,153.053
C07905=1091.254,258.421,-78.216,176.882,20.696,153.053
C07906=1091.248,258.172,-78.189,176.879,20.694,153.053
C07907=1091.242,257.923,-78.161,176.875,20.691,153.053
C07908=1091.236,257.676,-78.134,176.872,20.689,153.053
C07909=1091.231,257.427,-78.106,176.870,20.687,153.053
C07910=1091.225,257.178,-78.078,176.867,20.684,153.053
C07911=1091.219,256.930,-78.051,176.864,20.682,153.053
C07912=1091.214,256.682,-78.023,176.860,20.680,153.053
C07913=1091.208,256.433,-77.997,176.858,20.678,153.053
C07914=1091.202,256.185,-77.968,176.855,20.675,153.053
C07915=1091.197,255.936,-77.941,176.852,20.673,153.053
C07916=1091.192,255.688,-77.915,176.848,20.670,153.053
C07917=1091.186,255.439,-77.886,176.846,20.668,153.053
C07918=1091.180,255.191,-77.860,176.843,20.666,153.053
C07919=1091.174,254.943,-77.832,176.840,20.663,153.053
C07920=1091.169,254.694,-77.805,176.836,20.661,153.053
C07921=1091.163,254.446,-77.777,176.834,20.659,153.053
C07922=1091.157,254.197,-77.750,176.831,20.656,153.053
C07923=1091.152,253.948,-77.723,176.828,20.654,153.053
C07924=1091.146,253.701,-77.695,176.824,20.651,153.053
C07925=1091.141,253.452,-77.668,176.822,20.649,153.053
C07926=1091.136,253.203,-77.641,176.819,20.647,153.053
C07927=1091.129,252.955,-77.613,176.816,20.644,153.053
C07928=1091.124,252.706,-77.586,176.813,20.642,153.053
C07929=1091.118,252.458,-77.559,176.810,20.640,153.053
C07930=1091.113,252.209,-77.532,176.807,20.637,153.053
C07931=1091.107,251.961,-77.505,176.804,20.635,153.053
C07932=1091.102,251.713,-77.477,176.801,20.633,153.053
C07933=1091.096,251.464,-77.450,176.798,20.631,153.053
C07934=1091.090,251.215,-77.424,176.795,20.628,153.053
C07935=1091.085,250.967,-77.396,176.792,20.626,153.052
C07936=1091.079,250.719,-77.369,176.790,20.624,153.052
C07937=1091.074,250.470,-77.342,176.786,20.621,153.052
C07938=1091.068,250.222,-77.315,176.783,20.619,153.052
C07939=1091.060,249.852,-77.274,176.779,20.615,153.052
C07940=1091.052,249.483,-77.235,176.774,20.612,153.052
C07941=1091.043,249.115,-77.195,176.771,20.608,153.052
C07942=1091.035,248.746,-77.155,176.766,20.604,153.052
C07943=1091.030,248.497,-77.127,176.764,20.602,153.052
C07944=1091.024,248.249,-77.101,176.760,20.600,153.052
C07945=1091.019,248.000,-77.074,176.757,20.597,153.052
C07946=1091.013,247.752,-77.047,176.754,20.595,153.052
C07947=1091.008,247.503,-77.020,176.752,20.593,153.052
C07948=1091.002,247.254,-76.993,176.748,20.590,153.052
C07949=1090.996,247.006,-76.966,176.745,20.588,153.052
C07950=1090.990,246.758,-76.939,176.743,20.586,153.052
C07951=1090.985,246.509,-76.912,176.740,20.584,153.052
C07952=1090.980,246.261,-76.885,176.736,20.582,153.052
C07953=1090.974,246.012,-76.859,176.734,20.580,153.052
C07954=1090.968,245.763,-76.833,176.731,20.577,153.052
C07955=1090.963,245.515,-76.806,176.728,20.575,153.052
C07956=1090.958,245.266,-76.779,176.725,20.573,153.052
C07957=1090.952,245.018,-76.752,176.722,20.570,153.052
C07958=1090.946,244.770,-76.726,176.719,20.568,153.052
C07959=1090.940,244.521,-76.699,176.716,20.566,153.052
C07960=1090.935,244.273,-76.672,176.713,20.563,153.052
C07961=1090.930,244.024,-76.646,176.710,20.561,153.052
C07962=1090.924,243.775,-76.619,176.708,20.559,153.052
C07963=1090.918,243.527,-76.593,176.705,20.556,153.052
C07964=1090.912,243.278,-76.566,176.701,20.554,153.052
C07965=1090.907,243.030,-76.539,176.699,20.552,153.052
C07966=1090.902,242.781,-76.513,176.696,20.549,153.052
C07967=1090.896,242.532,-76.486,176.692,20.547,153.052
C07968=1090.890,242.284,-76.459,176.690,20.545,153.052
C07969=1090.885,242.036,-76.433,176.687,20.543,153.052
C07970=1090.879,241.787,-76.407,176.684,20.540,153.052
C07971=1090.873,241.538,-76.380,176.681,20.538,153.051
C07972=1090.868,241.290,-76.354,176.678,20.536,153.051
C07973=1090.862,241.041,-76.328,176.675,20.533,153.051
C07974=1090.856,240.793,-76.301,176.672,20.532,153.052
C07975=1090.851,240.544,-76.274,176.669,20.529,153.052
C07976=1090.845,240.295,-76.248,176.666,20.527,153.052
C07977=1090.839,240.047,-76.222,176.664,20.525,153.051
C07978=1090.834,239.798,-76.196,176.660,20.522,153.051
C07979=1090.828,239.550,-76.169,176.657,20.520,153.051
C07980=1090.822,239.301,-76.143,176.655,20.518,153.051
C07981=1090.817,239.052,-76.117,176.651,20.516,153.052
C07982=1090.811,238.804,-76.090,176.649,20.514,153.051
C07983=1090.805,238.555,-76.065,176.646,20.512,153.051
C07984=1090.799,238.307,-76.038,176.643,20.509,153.051
C07985=1090.794,238.058,-76.012,176.640,20.507,153.051
C07986=1090.788,237.810,-75.986,176.637,20.505,153.051
C07987=1090.783,237.561,-75.960,176.634,20.503,153.052
C07988=1090.777,237.313,-75.933,176.631,20.501,153.051
C07989=1090.772,237.064,-75.907,176.628,20.498,153.051
C07990=1090.766,236.816,-75.881,176.626,20.496,153.051
C07991=1090.758,236.440,-75.841,176.621,20.493,153.051
C07992=1090.749,236.064,-75.802,176.617,20.489,153.051
C07993=1090.740,235.688,-75.763,176.612,20.486,153.051
C07994=1090.732,235.312,-75.724,176.608,20.483,153.051
C07995=1090.726,235.064,-75.697,176.605,20.480,153.051
C07996=1090.721,234.815,-75.671,176.602,20.478,153.051
C07997=1090.715,234.566,-75.645,176.600,20.476,153.051
C07998=1090.710,234.317,-75.619,176.596,20.473,153.051
C07999=1090.705,234.069,-75.593,176.594,20.471,153.051
C08000=1090.699,233.820,-75.568,176.591,20.469,153.051
C08001=1090.693,233.572,-75.541,176.587,20.467,153.051
C08002=1090.687,233.323,-75.515,176.585,20.465,153.051
C08003=1090.682,233.074,-75.489,176.582,20.462,153.051
C08004=1090.676,232.826,-75.464,176.580,20.460,153.051
C08005=1090.671,232.578,-75.438,176.576,20.458,153.051
C08006=1090.665,232.329,-75.412,176.573,20.456,153.051
C08007=1090.660,232.080,-75.386,176.571,20.454,153.051
C08008=1090.653,231.831,-75.360,176.567,20.451,153.051
C08009=1090.648,231.583,-75.335,176.565,20.449,153.051
C08010=1090.643,231.334,-75.309,176.562,20.447,153.051
C08011=1090.637,231.086,-75.283,176.560,20.445,153.051
C08012=1090.631,230.837,-75.257,176.556,20.443,153.051
C08013=1090.626,230.588,-75.231,176.553,20.440,153.051
C08014=1090.620,230.340,-75.206,176.551,20.439,153.051
C08015=1090.615,230.091,-75.180,176.547,20.436,153.051
C08016=1090.609,229.842,-75.154,176.545,20.434,153.051
C08017=1090.603,229.593,-75.129,176.542,20.432,153.051
C08018=1090.598,229.345,-75.103,176.538,20.430,153.051
C08019=1090.592,229.096,-75.078,176.536,20.428,153.051
C08020=1090.586,228.847,-75.052,176.533,20.425,153.051
C08021=1090.580,228.599,-75.027,176.530,20.424,153.051
C08022=1090.575,228.350,-75.001,176.527,20.421,153.051
C08023=1090.569,228.102,-74.976,176.525,20.419,153.051
C08024=1090.564,227.853,-74.950,176.522,20.417,153.051
C08025=1090.558,227.605,-74.925,176.519,20.415,153.051
C08026=1090.552,227.356,-74.899,176.516,20.413,153.051
C08027=1090.546,227.107,-74.874,176.513,20.410,153.051
C08028=1090.541,226.858,-74.848,176.510,20.408,153.051
C08029=1090.535,226.610,-74.823,176.507,20.406,153.051
C08030=1090.530,226.361,-74.797,176.505,20.404,153.051
C08031=1090.524,226.112,-74.771,176.501,20.402,153.051
C08032=1090.519,225.864,-74.746,176.499,20.400,153.051
C08033=1090.512,225.615,-74.721,176.496,20.397,153.051
C08034=1090.507,225.366,-74.695,176.494,20.395,153.051
C08035=1090.502,225.118,-74.670,176.490,20.393,153.051
C08036=1090.496,224.869,-74.644,176.487,20.391,153.051
C08037=1090.490,224.620,-74.619,176.485,20.389,153.051
C08038=1090.485,224.372,-74.594,176.481,20.386,153.051
C08039=1090.479,224.123,-74.568,176.479,20.384,153.051
C08040=1090.474,223.874,-74.543,176.476,20.382,153.051
C08041=1090.468,223.626,-74.518,176.473,20.380,153.051
C08042=1090.463,223.377,-74.492,176.470,20.378,153.051
C08043=1090.454,222.992,-74.453,176.466,20.375,153.051
C08044=1090.445,222.608,-74.414,176.461,20.371,153.051
C08045=1090.437,222.224,-74.376,176.457,20.368,153.051
C08046=1090.428,221.839,-74.337,176.453,20.364,153.051
C08047=1090.422,221.590,-74.311,176.450,20.362,153.051
C08048=1090.417,221.342,-74.287,176.447,20.360,153.052
C08049=1090.411,221.093,-74.261,176.444,20.358,153.051
C08050=1090.405,220.845,-74.236,176.441,20.356,153.051
C08051=1090.400,220.595,-74.211,176.439,20.354,153.051
C08052=1090.394,220.347,-74.186,176.436,20.352,153.052
C08053=1090.389,220.098,-74.162,176.433,20.350,153.052
C08054=1090.382,219.850,-74.136,176.430,20.347,153.052
C08055=1090.378,219.601,-74.111,176.428,20.345,153.051
C08056=1090.372,219.352,-74.086,176.424,20.343,153.052
C08057=1090.366,219.104,-74.061,176.422,20.341,153.052
C08058=1090.360,218.855,-74.036,176.419,20.339,153.052
C08059=1090.354,218.606,-74.011,176.416,20.337,153.052
C08060=1090.349,218.357,-73.986,176.413,20.335,153.052
C08061=1090.343,218.108,-73.961,176.411,20.333,153.052
C08062=1090.338,217.860,-73.937,176.408,20.330,153.052
C08063=1090.332,217.611,-73.911,176.405,20.328,153.052
C08064=1090.326,217.363,-73.887,176.402,20.326,153.052
C08065=1090.321,217.114,-73.861,176.399,20.324,153.052
C08066=1090.316,216.865,-73.837,176.396,20.322,153.052
C08067=1090.310,216.616,-73.812,176.394,20.320,153.052
C08068=1090.304,216.368,-73.787,176.391,20.318,153.052
C08069=1090.298,216.119,-73.763,176.388,20.316,153.052
C08070=1090.293,215.871,-73.738,176.385,20.314,153.052
C08071=1090.287,215.622,-73.713,176.383,20.312,153.052
C08072=1090.282,215.372,-73.688,176.379,20.310,153.052
C08073=1090.277,215.124,-73.663,176.377,20.308,153.052
C08074=1090.271,214.875,-73.639,176.374,20.305,153.052
C08075=1090.265,214.627,-73.614,176.371,20.303,153.052
C08076=1090.259,214.378,-73.589,176.368,20.301,153.052
C08077=1090.254,214.129,-73.565,176.366,20.299,153.052
C08078=1090.249,213.881,-73.541,176.362,20.297,153.052
C08079=1090.242,213.632,-73.515,176.360,20.295,153.052
C08080=1090.237,213.383,-73.491,176.358,20.293,153.052
C08081=1090.231,213.134,-73.466,176.354,20.291,153.052
C08082=1090.226,212.886,-73.442,176.352,20.289,153.052
C08083=1090.220,212.637,-73.417,176.349,20.286,153.052
C08084=1090.214,212.388,-73.392,176.347,20.284,153.052
C08085=1090.209,212.140,-73.368,176.343,20.282,153.052
C08086=1090.203,211.890,-73.344,176.341,20.280,153.052
C08087=1090.198,211.642,-73.319,176.338,20.278,153.052
C08088=1090.192,211.393,-73.295,176.335,20.276,153.052
C08089=1090.186,211.145,-73.270,176.332,20.274,153.052
C08090=1090.181,210.896,-73.246,176.330,20.272,153.052
C08091=1090.175,210.647,-73.221,176.326,20.269,153.052
C08092=1090.170,210.398,-73.197,176.324,20.267,153.052
C08093=1090.165,210.150,-73.172,176.322,20.266,153.052
C08094=1090.159,209.900,-73.148,176.318,20.263,153.052
C08095=1090.150,209.520,-73.110,176.314,20.260,153.052
C08096=1090.142,209.139,-73.073,176.310,20.257,153.052
C08097=1090.133,208.759,-73.036,176.305,20.254,153.052
C08098=1090.124,208.378,-72.999,176.302,20.250,153.052
C08099=1090.101,207.356,-72.900,176.233,20.217,153.056
C08100=1090.096,207.107,-72.876,176.231,20.216,153.056
C08101=1090.090,206.859,-72.853,176.228,20.215,153.057
C08102=1090.085,206.610,-72.829,176.225,20.213,153.057
C08103=1090.079,206.361,-72.804,176.222,20.212,153.057
C08104=1090.073,206.112,-72.781,176.219,20.211,153.057
C08105=1090.068,205.863,-72.757,176.216,20.210,153.058
C08106=1090.062,205.615,-72.734,176.213,20.209,153.058
C08107=1090.057,205.366,-72.709,176.211,20.208,153.058
C08108=1090.052,205.117,-72.686,176.208,20.206,153.058
C08109=1090.045,204.868,-72.662,176.204,20.205,153.058
C08110=1090.040,204.619,-72.637,176.202,20.204,153.059
C08111=1090.034,204.371,-72.615,176.199,20.203,153.059
C08112=1090.029,204.122,-72.590,176.196,20.202,153.059
C08113=1090.024,203.873,-72.567,176.193,20.200,153.059
C08114=1090.018,203.624,-72.543,176.191,20.199,153.060
C08115=1090.012,203.376,-72.519,176.187,20.198,153.060
C08116=1090.006,203.126,-72.496,176.184,20.197,153.060
C08117=1090.001,202.878,-72.471,176.182,20.195,153.060
C08118=1089.995,202.629,-72.448,176.179,20.194,153.060
C08119=1089.990,202.380,-72.424,176.176,20.193,153.061
C08120=1089.984,202.131,-72.401,176.173,20.192,153.061
C08121=1089.979,201.883,-72.377,176.171,20.191,153.061
C08122=1089.973,201.634,-72.354,176.167,20.189,153.062
C08123=1089.966,201.385,-72.330,176.164,20.188,153.062
C08124=1089.961,201.136,-72.306,176.161,20.187,153.062
C08125=1089.955,200.887,-72.283,176.159,20.186,153.062
C08126=1089.950,200.638,-72.260,176.156,20.185,153.062
C08127=1089.945,200.389,-72.236,176.153,20.184,153.063
C08128=1089.939,200.141,-72.213,176.150,20.183,153.063
C08129=1089.934,199.892,-72.189,176.147,20.181,153.063
C08130=1089.928,199.643,-72.165,176.144,20.180,153.063
C08131=1089.921,199.394,-72.142,176.141,20.179,153.064
C08132=1089.916,199.145,-72.118,176.139,20.178,153.064
C08133=1089.910,198.896,-72.095,176.136,20.177,153.064
C08134=1089.904,198.647,-72.072,176.133,20.176,153.064
C08135=1089.899,198.398,-72.048,176.130,20.175,153.065
C08136=1089.893,198.150,-72.025,176.128,20.174,153.065
C08137=1089.888,197.901,-72.002,176.124,20.172,153.065
C08138=1089.882,197.652,-71.979,176.121,20.171,153.065
C08139=1089.877,197.404,-71.955,176.119,20.170,153.065
C08140=1089.871,197.155,-71.932,176.116,20.169,153.066
C08141=1089.865,196.906,-71.909,176.113,20.168,153.066
C08142=1089.860,196.657,-71.884,176.110,20.166,153.066
C08143=1089.854,196.408,-71.861,176.108,20.165,153.066
C08144=1089.848,196.159,-71.838,176.105,20.164,153.067
C08145=1089.843,195.911,-71.816,176.102,20.163,153.067
C08146=1089.838,195.661,-71.792,176.099,20.162,153.067
C08147=1089.832,195.413,-71.768,176.096,20.160,153.067
C08148=1089.826,195.164,-71.745,176.093,20.159,153.067
C08149=1089.821,194.915,-71.722,176.090,20.158,153.068
C08150=1089.815,194.666,-71.699,176.088,20.157,153.068
C08151=1089.809,194.417,-71.676,176.085,20.156,153.068
C08152=1089.804,194.168,-71.653,176.082,20.155,153.068
C08153=1089.798,193.920,-71.629,176.079,20.154,153.069
C08154=1089.793,193.671,-71.606,176.077,20.152,153.069
C08155=1089.787,193.422,-71.583,176.074,20.151,153.069
C08156=1089.781,193.173,-71.560,176.071,20.150,153.069
C08157=1089.776,192.924,-71.537,176.068,20.149,153.069
C08158=1089.771,192.675,-71.513,176.065,20.147,153.070
C08159=1089.765,192.426,-71.490,176.062,20.146,153.070
C08160=1089.758,192.150,-71.465,176.060,20.145,153.070
C08161=1089.752,191.873,-71.439,176.057,20.144,153.070
C08162=1089.746,191.596,-71.414,176.053,20.142,153.070
C08163=1089.740,191.319,-71.388,176.051,20.141,153.071
C08164=1089.734,191.070,-71.365,176.048,20.140,153.071
C08165=1089.729,190.821,-71.342,176.045,20.138,153.071
C08166=1089.724,190.572,-71.319,176.042,20.137,153.071
C08167=1089.718,190.323,-71.296,176.039,20.136,153.072
C08168=1089.712,190.074,-71.273,176.036,20.134,153.072
C08169=1089.707,189.825,-71.250,176.033,20.133,153.072
C08170=1089.702,189.577,-71.227,176.031,20.132,153.072
C08171=1089.696,189.328,-71.204,176.028,20.131,153.072
C08172=1089.691,189.079,-71.181,176.025,20.130,153.073
C08173=1089.685,188.830,-71.158,176.023,20.128,153.073
C08174=1089.679,188.581,-71.135,176.020,20.127,153.073
C08175=1089.673,188.332,-71.112,176.017,20.126,153.073
C08176=1089.669,188.084,-71.090,176.015,20.125,153.073
C08177=1089.664,187.834,-71.067,176.012,20.124,153.074
C08178=1089.658,187.585,-71.044,176.009,20.122,153.074
C08179=1089.652,187.337,-71.021,176.006,20.121,153.074
C08180=1089.646,187.088,-70.998,176.004,20.120,153.074
C08181=1089.641,186.840,-70.975,176.001,20.119,153.074
C08182=1089.636,186.590,-70.953,175.998,20.118,153.075
C08183=1089.630,186.341,-70.930,175.996,20.116,153.075
C08184=1089.624,186.092,-70.907,175.993,20.115,153.075
C08185=1089.619,185.843,-70.884,175.990,20.114,153.075
C08186=1089.614,185.595,-70.862,175.988,20.113,153.075
C08187=1089.609,185.345,-70.839,175.984,20.111,153.076
C08188=1089.603,185.096,-70.816,175.981,20.110,153.076
C08189=1089.597,184.848,-70.794,175.979,20.109,153.076
C08190=1089.591,184.599,-70.771,175.976,20.108,153.076
C08191=1089.586,184.350,-70.749,175.973,20.106,153.076
C08192=1089.580,184.101,-70.726,175.971,20.105,153.077
C08193=1089.574,183.853,-70.704,175.968,20.104,153.077
C08194=1089.569,183.603,-70.681,175.965,20.103,153.077
C08195=1089.563,183.354,-70.658,175.962,20.102,153.077
C08196=1089.557,183.105,-70.635,175.960,20.101,153.077
C08197=1089.551,182.856,-70.614,175.957,20.100,153.078
C08198=1089.546,182.608,-70.591,175.954,20.099,153.078
C08199=1089.540,182.359,-70.568,175.952,20.097,153.078
C08200=1089.535,182.109,-70.546,175.949,20.096,153.078
C08201=1089.528,181.861,-70.524,175.946,20.095,153.079
C08202=1089.523,181.611,-70.501,175.943,20.094,153.079
C08203=1089.518,181.363,-70.479,175.941,20.093,153.079
C08204=1089.512,181.114,-70.456,175.938,20.092,153.079
C08205=1089.506,180.865,-70.434,175.935,20.090,153.079
C08206=1089.500,180.616,-70.411,175.933,20.089,153.080
C08207=1089.495,180.367,-70.389,175.930,20.088,153.080
C08208=1089.489,180.119,-70.367,175.927,20.086,153.080
C08209=1089.483,179.869,-70.345,175.924,20.085,153.080
C08210=1089.478,179.620,-70.322,175.922,20.084,153.081
C08211=1089.471,179.371,-70.300,175.919,20.083,153.081
C08212=1089.466,179.123,-70.278,175.916,20.082,153.081
C08213=1089.461,178.873,-70.256,175.913,20.081,153.081
C08214=1089.454,178.625,-70.233,175.911,20.079,153.081
C08215=1089.449,178.375,-70.211,175.908,20.078,153.082
C08216=1089.444,178.127,-70.188,175.906,20.077,153.082
C08217=1089.438,177.878,-70.167,175.903,20.076,153.082
C08218=1089.432,177.628,-70.145,175.900,20.075,153.082
C08219=1089.426,177.380,-70.122,175.897,20.073,153.082
C08220=1089.421,177.131,-70.100,175.896,20.073,153.082
C08221=1089.415,176.882,-70.077,175.893,20.071,153.083
C08222=1089.410,176.633,-70.055,175.890,20.070,153.083
C08223=1089.404,176.384,-70.034,175.887,20.069,153.083
C08224=1089.398,176.107,-70.009,175.884,20.067,153.083
C08225=1089.391,175.830,-69.984,175.881,20.066,153.084
C08226=1089.385,175.552,-69.959,175.879,20.065,153.084
C08227=1089.378,175.275,-69.935,175.875,20.063,153.084
C08228=1089.374,175.026,-69.913,175.872,20.062,153.084
C08229=1089.368,174.778,-69.890,175.870,20.061,153.084
C08230=1089.362,174.528,-69.868,175.867,20.060,153.085
C08231=1089.357,174.280,-69.846,175.865,20.059,153.085
C08232=1089.351,174.030,-69.825,175.862,20.058,153.085
C08233=1089.346,173.782,-69.802,175.860,20.056,153.085
C08234=1089.340,173.533,-69.780,175.857,20.055,153.085
C08235=1089.334,173.283,-69.758,175.854,20.054,153.085
C08236=1089.329,173.035,-69.737,175.852,20.053,153.086
C08237=1089.323,172.786,-69.714,175.849,20.051,153.086
C08238=1089.318,172.537,-69.692,175.846,20.050,153.086
C08239=1089.312,172.288,-69.671,175.844,20.049,153.086
C08240=1089.306,172.038,-69.648,175.841,20.048,153.086
C08241=1089.301,171.790,-69.627,175.838,20.046,153.086
C08242=1089.295,171.540,-69.605,175.836,20.045,153.087
C08243=1089.290,171.292,-69.582,175.833,20.044,153.087
C08244=1089.284,171.043,-69.561,175.831,20.042,153.087
C08245=1089.279,170.794,-69.539,175.828,20.041,153.087
C08246=1089.273,170.545,-69.517,175.825,20.040,153.087
C08247=1089.268,170.295,-69.495,175.822,20.039,153.088
C08248=1089.262,170.047,-69.474,175.820,20.037,153.088
C08249=1089.257,169.797,-69.451,175.818,20.036,153.088
C08250=1089.251,169.549,-69.430,175.815,20.035,153.088
C08251=1089.246,169.299,-69.408,175.813,20.034,153.088
C08252=1089.240,169.051,-69.387,175.810,20.033,153.088
C08253=1089.234,168.802,-69.364,175.807,20.031,153.089
C08254=1089.229,168.554,-69.343,175.805,20.030,153.089
C08255=1089.223,168.304,-69.320,175.802,20.029,153.089
C08256=1089.218,168.056,-69.299,175.800,20.027,153.089
C08257=1089.212,167.806,-69.277,175.797,20.026,153.089
C08258=1089.207,167.558,-69.256,175.794,20.025,153.089
C08259=1089.201,167.308,-69.233,175.792,20.023,153.090
C08260=1089.196,167.059,-69.212,175.789,20.022,153.090
C08261=1089.190,166.810,-69.190,175.786,20.021,153.090
C08262=1089.185,166.561,-69.169,175.784,20.019,153.090
C08263=1089.180,166.312,-69.147,175.782,20.018,153.090
C08264=1089.174,166.063,-69.126,175.779,20.017,153.090
C08265=1089.169,165.814,-69.104,175.777,20.016,153.091
C08266=1089.163,165.565,-69.082,175.774,20.014,153.091
C08267=1089.158,165.316,-69.061,175.771,20.013,153.091
C08268=1089.152,165.067,-69.039,175.769,20.012,153.091
C08269=1089.147,164.818,-69.017,175.766,20.010,153.091
C08270=1089.142,164.569,-68.996,175.764,20.009,153.091
C08271=1089.136,164.320,-68.974,175.761,20.008,153.092
C08272=1089.131,164.071,-68.953,175.758,20.006,153.092
C08273=1089.125,163.822,-68.931,175.757,20.005,153.092
C08274=1089.119,163.573,-68.910,175.754,20.004,153.092
C08275=1089.115,163.324,-68.888,175.751,20.003,153.092
C08276=1089.108,163.075,-68.866,175.749,20.001,153.092
C08277=1089.104,162.826,-68.845,175.746,20.000,153.092
C08278=1089.098,162.577,-68.824,175.744,19.998,153.092
C08279=1089.092,162.328,-68.802,175.741,19.997,153.093
C08280=1089.087,162.079,-68.780,175.738,19.996,153.093
C08281=1089.081,161.829,-68.760,175.736,19.994,153.093
C08282=1089.077,161.580,-68.738,175.733,19.993,153.093
C08283=1089.071,161.332,-68.716,175.731,19.992,153.093
C08284=1089.065,161.083,-68.695,175.729,19.991,153.093
C08285=1089.060,160.834,-68.674,175.726,19.989,153.094
C08286=1089.054,160.584,-68.653,175.723,19.988,153.094
C08287=1089.048,160.336,-68.631,175.721,19.987,153.094
C08288=1089.042,160.056,-68.608,175.718,19.985,153.094
C08289=1089.036,159.777,-68.584,175.716,19.984,153.094
C08290=1089.029,159.496,-68.560,175.712,19.982,153.094
C08291=1089.023,159.217,-68.536,175.710,19.981,153.095
C08292=1089.017,158.968,-68.514,175.707,19.980,153.095
C08293=1089.012,158.719,-68.494,175.704,19.978,153.095
C08294=1089.006,158.470,-68.472,175.703,19.977,153.095
C08295=1089.001,158.221,-68.451,175.700,19.976,153.095
C08296=1088.995,157.972,-68.430,175.697,19.975,153.095
C08297=1088.989,157.723,-68.408,175.695,19.973,153.096
C08298=1088.984,157.474,-68.388,175.692,19.972,153.096
C08299=1088.978,157.225,-68.367,175.689,19.971,153.096
C08300=1088.973,156.975,-68.345,175.687,19.969,153.096
C08301=1088.967,156.727,-68.324,175.685,19.968,153.096
C08302=1088.962,156.477,-68.303,175.682,19.967,153.096
C08303=1088.956,156.228,-68.282,175.680,19.965,153.096
C08304=1088.951,155.979,-68.261,175.677,19.964,153.097
C08305=1088.945,155.731,-68.240,175.675,19.963,153.097
C08306=1088.939,155.481,-68.219,175.672,19.961,153.097
C08307=1088.934,155.232,-68.198,175.669,19.960,153.097
C08308=1088.928,154.983,-68.177,175.668,19.959,153.097
C08309=1088.922,154.734,-68.155,175.665,19.958,153.097
C08310=1088.917,154.485,-68.135,175.662,19.956,153.097
C08311=1088.911,154.236,-68.114,175.660,19.955,153.098
C08312=1088.906,153.987,-68.093,175.657,19.954,153.098
C08313=1088.900,153.738,-68.071,175.655,19.952,153.098
C08314=1088.895,153.489,-68.051,175.653,19.951,153.098
C08315=1088.890,153.240,-68.030,175.650,19.950,153.098
C08316=1088.883,152.991,-68.009,175.648,19.948,153.098
C08317=1088.877,152.742,-67.989,175.645,19.947,153.099
C08318=1088.872,152.493,-67.967,175.642,19.946,153.099
C08319=1088.866,152.243,-67.947,175.640,19.944,153.099
C08320=1088.861,151.994,-67.926,175.638,19.943,153.099
C08321=1088.855,151.746,-67.905,175.636,19.942,153.099
C08322=1088.850,151.497,-67.884,175.633,19.940,153.099
C08323=1088.844,151.247,-67.863,175.630,19.939,153.099
C08324=1088.838,150.998,-67.842,175.628,19.938,153.099
C08325=1088.833,150.749,-67.821,175.625,19.936,153.100
C08326=1088.828,150.500,-67.801,175.623,19.935,153.100
C08327=1088.822,150.251,-67.779,175.621,19.934,153.100
C08328=1088.816,150.002,-67.759,175.618,19.932,153.100
C08329=1088.811,149.753,-67.739,175.616,19.931,153.100
C08330=1088.805,149.504,-67.718,175.613,19.929,153.100
C08331=1088.800,149.255,-67.697,175.610,19.928,153.100
C08332=1088.794,149.005,-67.676,175.609,19.927,153.101
C08333=1088.789,148.756,-67.655,175.606,19.926,153.101
C08334=1088.783,148.507,-67.635,175.604,19.924,153.101
C08335=1088.777,148.258,-67.615,175.601,19.923,153.101
C08336=1088.772,148.010,-67.594,175.598,19.921,153.101
C08337=1088.766,147.762,-67.573,175.597,19.920,153.101
C08338=1088.760,147.514,-67.553,175.594,19.919,153.101
C08339=1088.755,147.267,-67.532,175.591,19.918,153.101
C08340=1088.749,147.018,-67.512,175.589,19.916,153.102
C08341=1088.743,146.770,-67.491,175.586,19.915,153.102
C08342=1088.738,146.522,-67.471,175.585,19.914,153.102
C08343=1088.732,146.274,-67.450,175.582,19.912,153.102
C08344=1088.727,146.025,-67.429,175.580,19.911,153.102
C08345=1088.721,145.776,-67.409,175.577,19.909,153.102
C08346=1088.715,145.527,-67.389,175.574,19.908,153.102
C08347=1088.710,145.278,-67.368,175.573,19.907,153.102
C08348=1088.705,145.029,-67.348,175.570,19.905,153.103
C08349=1088.698,144.779,-67.327,175.567,19.904,153.103
C08350=1088.693,144.530,-67.307,175.565,19.903,153.103
C08351=1088.688,144.281,-67.286,175.563,19.902,153.103
C08352=1088.681,144.004,-67.264,175.560,19.900,153.103
C08353=1088.675,143.726,-67.241,175.557,19.898,153.103
C08354=1088.669,143.448,-67.218,175.555,19.897,153.103
C08355=1088.662,143.171,-67.195,175.552,19.895,153.104
C08356=1088.657,142.921,-67.175,175.549,19.894,153.104
C08357=1088.652,142.672,-67.154,175.548,19.893,153.104
C08358=1088.646,142.424,-67.134,175.545,19.891,153.104
C08359=1088.640,142.174,-67.113,175.543,19.890,153.104
C08360=1088.635,141.925,-67.093,175.540,19.888,153.104
C08361=1088.629,141.676,-67.073,175.538,19.887,153.104
C08362=1088.624,141.427,-67.052,175.536,19.886,153.104
C08363=1088.618,141.178,-67.032,175.533,19.884,153.104
C08364=1088.613,140.928,-67.012,175.531,19.883,153.105
C08365=1088.607,140.679,-66.992,175.528,19.881,153.105
C08366=1088.601,140.430,-66.972,175.526,19.880,153.105
C08367=1088.596,140.181,-66.951,175.524,19.879,153.105
C08368=1088.590,139.932,-66.931,175.521,19.877,153.105
C08369=1088.585,139.683,-66.911,175.519,19.876,153.105
C08370=1088.579,139.434,-66.891,175.516,19.874,153.105
C08371=1088.573,139.184,-66.870,175.515,19.873,153.105
C08372=1088.567,138.935,-66.851,175.512,19.872,153.105
C08373=1088.562,138.686,-66.830,175.509,19.870,153.106
C08374=1088.556,138.437,-66.810,175.507,19.868,153.106
C08375=1088.551,138.188,-66.790,175.505,19.867,153.106
C08376=1088.545,137.939,-66.770,175.503,19.866,153.106
C08377=1088.540,137.689,-66.750,175.500,19.864,153.106
C08378=1088.534,137.441,-66.730,175.498,19.863,153.106
C08379=1088.529,137.191,-66.709,175.496,19.862,153.106
C08380=1088.523,136.943,-66.689,175.494,19.860,153.106
C08381=1088.517,136.694,-66.669,175.491,19.859,153.106
C08382=1088.512,136.444,-66.650,175.488,19.857,153.107
C08383=1088.506,136.195,-66.630,175.487,19.856,153.107
C08384=1088.500,135.946,-66.609,175.484,19.855,153.107
C08385=1088.495,135.697,-66.590,175.482,19.853,153.107
C08386=1088.489,135.448,-66.569,175.479,19.852,153.107
C08387=1088.483,135.199,-66.549,175.477,19.851,153.107
C08388=1088.477,134.950,-66.529,175.475,19.849,153.107
C08389=1088.473,134.700,-66.510,175.472,19.847,153.107
C08390=1088.467,134.451,-66.490,175.470,19.846,153.107
C08391=1088.461,134.202,-66.469,175.468,19.845,153.107
C08392=1088.456,133.953,-66.450,175.466,19.843,153.107
C08393=1088.450,133.704,-66.430,175.463,19.842,153.108
C08394=1088.445,133.454,-66.410,175.461,19.840,153.108
C08395=1088.439,133.206,-66.390,175.459,19.839,153.108
C08396=1088.433,132.956,-66.370,175.457,19.837,153.108
C08397=1088.428,132.707,-66.350,175.454,19.836,153.108
C08398=1088.422,132.458,-66.330,175.452,19.835,153.108
C08399=1088.417,132.208,-66.310,175.450,19.833,153.108
C08400=1088.411,131.960,-66.291,175.447,19.832,153.108
C08401=1088.405,131.711,-66.271,175.445,19.830,153.108
C08402=1088.399,131.461,-66.251,175.443,19.829,153.108
C08403=1088.393,131.213,-66.231,175.440,19.828,153.109
C08404=1088.388,130.963,-66.212,175.438,19.826,153.109
C08405=1088.382,130.714,-66.192,175.436,19.824,153.109
C08406=1088.376,130.465,-66.172,175.434,19.823,153.109
C08407=1088.370,130.216,-66.152,175.431,19.822,153.109
C08408=1088.365,129.966,-66.133,175.429,19.820,153.109
C08409=1088.359,129.717,-66.113,175.427,19.819,153.109
C08410=1088.354,129.468,-66.093,175.424,19.818,153.109
C08411=1088.348,129.219,-66.073,175.422,19.816,153.109
C08412=1088.342,128.969,-66.054,175.420,19.814,153.109
C08413=1088.336,128.721,-66.034,175.418,19.813,153.109
C08414=1088.330,128.471,-66.015,175.415,19.812,153.110
C08415=1088.325,128.222,-65.996,175.413,19.810,153.110
C08416=1088.319,127.945,-65.974,175.410,19.809,153.110
C08417=1088.312,127.667,-65.952,175.408,19.807,153.110
C08418=1088.306,127.389,-65.930,175.405,19.805,153.110
C08419=1088.299,127.111,-65.908,175.403,19.804,153.110
C08420=1088.294,126.862,-65.888,175.401,19.803,153.110
C08421=1088.289,126.612,-65.869,175.399,19.801,153.110
C08422=1088.283,126.363,-65.849,175.396,19.799,153.110
C08423=1088.277,126.114,-65.829,175.394,19.798,153.110
C08424=1088.272,125.865,-65.811,175.392,19.797,153.111
C08425=1088.266,125.616,-65.791,175.389,19.795,153.111
C08426=1088.260,125.367,-65.771,175.387,19.794,153.111
C08427=1088.254,125.117,-65.752,175.385,19.792,153.111
C08428=1088.249,124.868,-65.733,175.383,19.791,153.111
C08429=1088.243,124.619,-65.714,175.380,19.789,153.111
C08430=1088.238,124.369,-65.693,175.379,19.788,153.111
C08431=1088.233,124.121,-65.674,175.376,19.786,153.111
C08432=1088.227,123.871,-65.655,175.374,19.785,153.111
C08433=1088.221,123.623,-65.635,175.371,19.783,153.111
C08434=1088.215,123.373,-65.616,175.370,19.782,153.111
C08435=1088.210,123.124,-65.597,175.367,19.780,153.111
C08436=1088.204,122.874,-65.577,175.365,19.779,153.112
C08437=1088.199,122.625,-65.558,175.363,19.777,153.111
C08438=1088.193,122.377,-65.538,175.361,19.776,153.112
C08439=1088.187,122.127,-65.519,175.358,19.774,153.112
C08440=1088.181,121.878,-65.500,175.357,19.773,153.112
C08441=1088.176,121.628,-65.481,175.354,19.771,153.112
C08442=1088.171,121.380,-65.462,175.351,19.770,153.112
C08443=1088.165,121.131,-65.442,175.350,19.768,153.112
C08444=1088.159,120.881,-65.423,175.347,19.767,153.112
C08445=1088.153,120.632,-65.403,175.345,19.765,153.112
C08446=1088.148,120.383,-65.384,175.343,19.764,153.112
C08447=1088.143,120.134,-65.365,175.341,19.762,153.112
C08448=1088.137,119.884,-65.346,175.339,19.760,153.112
C08449=1088.131,119.635,-65.327,175.337,19.759,153.112
C08450=1088.125,119.385,-65.308,175.334,19.758,153.112
C08451=1088.120,119.137,-65.289,175.332,19.756,153.112
C08452=1088.115,118.887,-65.269,175.330,19.755,153.112
C08453=1088.109,118.639,-65.249,175.328,19.753,153.112
C08454=1088.104,118.390,-65.231,175.325,19.751,153.113
C08455=1088.098,118.140,-65.211,175.324,19.750,153.113
C08456=1088.092,117.891,-65.192,175.321,19.748,153.113
C08457=1088.087,117.641,-65.173,175.319,19.747,153.113
C08458=1088.081,117.393,-65.154,175.317,19.745,153.113
C08459=1088.076,117.143,-65.135,175.315,19.744,153.113
C08460=1088.070,116.894,-65.115,175.313,19.742,153.113
C08461=1088.065,116.645,-65.097,175.311,19.741,153.113
C08462=1088.059,116.396,-65.077,175.308,19.739,153.113
C08463=1088.054,116.146,-65.058,175.306,19.737,153.113
C08464=1088.049,115.898,-65.039,175.304,19.736,153.113
C08465=1088.043,115.648,-65.020,175.302,19.734,153.113
C08466=1088.037,115.398,-65.001,175.300,19.732,153.113
C08467=1088.032,115.149,-64.983,175.298,19.731,153.113
C08468=1088.026,114.900,-64.964,175.296,19.729,153.113
C08469=1088.020,114.651,-64.945,175.293,19.728,153.113
C08470=1088.015,114.402,-64.926,175.292,19.726,153.113
C08471=1088.010,114.153,-64.907,175.289,19.725,153.113
C08472=1088.004,113.903,-64.887,175.287,19.723,153.113
C08473=1087.999,113.654,-64.868,175.285,19.722,153.113
C08474=1087.992,113.405,-64.850,175.283,19.720,153.113
C08475=1087.987,113.155,-64.831,175.280,19.718,153.114
C08476=1087.981,112.906,-64.812,175.279,19.717,153.114
C08477=1087.976,112.657,-64.793,175.276,19.715,153.114
C08478=1087.970,112.408,-64.775,175.274,19.713,153.114
C08479=1087.964,112.159,-64.755,175.272,19.712,153.114
C08480=1087.958,111.880,-64.735,175.270,19.710,153.114
C08481=1087.952,111.603,-64.714,175.267,19.709,153.114
C08482=1087.946,111.325,-64.693,175.265,19.707,153.114
C08483=1087.939,111.047,-64.672,175.262,19.705,153.114
C08484=1087.934,110.798,-64.653,175.260,19.703,153.114
C08485=1087.928,110.549,-64.634,175.258,19.702,153.114
C08486=1087.922,110.299,-64.616,175.256,19.700,153.114
C08487=1087.917,110.050,-64.597,175.254,19.699,153.114
C08488=1087.910,109.801,-64.578,175.252,19.697,153.114
C08489=1087.905,109.552,-64.559,175.249,19.696,153.114
C08490=1087.900,109.302,-64.541,175.248,19.694,153.114
C08491=1087.893,109.053,-64.522,175.245,19.693,153.114
C08492=1087.888,108.804,-64.503,175.243,19.691,153.114
C08493=1087.883,108.554,-64.485,175.241,19.690,153.114
C08494=1087.877,108.305,-64.466,175.239,19.688,153.114
C08495=1087.871,108.057,-64.447,175.237,19.686,153.115
C08496=1087.865,107.807,-64.429,175.235,19.685,153.114
C08497=1087.860,107.557,-64.410,175.233,19.683,153.114
C08498=1087.854,107.309,-64.392,175.231,19.682,153.115
C08499=1087.848,107.059,-64.373,175.229,19.680,153.115
C08500=1087.843,106.810,-64.354,175.226,19.678,153.115
C08501=1087.837,106.561,-64.336,175.225,19.677,153.115
C08502=1087.832,106.311,-64.317,175.222,19.675,153.115
C08503=1087.826,106.063,-64.299,175.221,19.674,153.115
C08504=1087.820,105.813,-64.280,175.218,19.672,153.115
C08505=1087.815,105.564,-64.262,175.216,19.670,153.115
C08506=1087.809,105.314,-64.244,175.214,19.669,153.115
C08507=1087.804,105.065,-64.225,175.212,19.667,153.115
C08508=1087.798,104.816,-64.206,175.210,19.665,153.115
C08509=1087.793,104.567,-64.188,175.208,19.664,153.115
C08510=1087.786,104.318,-64.169,175.206,19.662,153.115
C08511=1087.781,104.068,-64.151,175.204,19.661,153.115
C08512=1087.775,103.819,-64.132,175.202,19.659,153.115
C08513=1087.770,103.569,-64.114,175.199,19.657,153.115
C08514=1087.764,103.321,-64.096,175.198,19.656,153.115
C08515=1087.759,103.071,-64.077,175.195,19.654,153.115
C08516=1087.753,102.822,-64.059,175.194,19.653,153.115
C08517=1087.747,102.572,-64.040,175.191,19.651,153.115
C08518=1087.742,102.324,-64.022,175.189,19.649,153.115
C08519=1087.736,102.074,-64.003,175.187,19.648,153.115
C08520=1087.731,101.825,-63.986,175.185,19.646,153.115
C08521=1087.725,101.575,-63.967,175.184,19.644,153.115
C08522=1087.720,101.326,-63.949,175.181,19.643,153.115
C08523=1087.714,101.077,-63.930,175.179,19.641,153.115
C08524=1087.708,100.828,-63.912,175.177,19.639,153.115
C08525=1087.702,100.579,-63.894,175.175,19.638,153.115
C08526=1087.697,100.329,-63.875,175.173,19.636,153.115
C08527=1087.691,100.080,-63.857,175.171,19.634,153.115
C08528=1087.685,99.831,-63.839,175.168,19.633,153.115
C08529=1087.680,99.581,-63.821,175.167,19.631,153.115
C08530=1087.674,99.332,-63.803,175.165,19.629,153.115
C08531=1087.668,99.083,-63.784,175.163,19.628,153.115
C08532=1087.663,98.834,-63.766,175.161,19.626,153.115
C08533=1087.657,98.584,-63.748,175.159,19.625,153.115
C08534=1087.651,98.336,-63.730,175.157,19.623,153.115
C08535=1087.646,98.085,-63.712,175.154,19.621,153.115
C08536=1087.640,97.836,-63.694,175.153,19.620,153.115
C08537=1087.634,97.587,-63.675,175.150,19.618,153.116
C08538=1087.629,97.338,-63.657,175.149,19.617,153.115
C08539=1087.623,97.088,-63.639,175.147,19.615,153.115
C08540=1087.617,96.840,-63.621,175.144,19.613,153.115
C08541=1087.612,96.591,-63.603,175.143,19.612,153.116
C08542=1087.606,96.341,-63.585,175.140,19.610,153.116
C08543=1087.601,96.092,-63.567,175.139,19.608,153.115
C08544=1087.594,95.814,-63.547,175.136,19.606,153.115
C08545=1087.588,95.536,-63.527,175.134,19.604,153.115
C08546=1087.581,95.258,-63.507,175.132,19.603,153.116
C08547=1087.575,94.980,-63.487,175.129,19.601,153.116
C08548=1087.570,94.731,-63.469,175.128,19.599,153.116
C08549=1087.564,94.481,-63.451,175.126,19.597,153.116
C08550=1087.558,94.233,-63.432,175.124,19.596,153.115
C08551=1087.552,93.983,-63.414,175.122,19.594,153.116
C08552=1087.547,93.734,-63.397,175.119,19.592,153.116
C08553=1087.542,93.484,-63.379,175.118,19.591,153.116
C08554=1087.536,93.235,-63.361,175.115,19.589,153.116
C08555=1087.530,92.986,-63.343,175.114,19.587,153.115
C08556=1087.525,92.737,-63.326,175.112,19.585,153.115
C08557=1087.519,92.487,-63.306,175.110,19.584,153.116
C08558=1087.514,92.238,-63.289,175.108,19.582,153.116
C08559=1087.508,91.989,-63.271,175.105,19.580,153.116
C08560=1087.502,91.739,-63.253,175.104,19.578,153.116
C08561=1087.496,91.490,-63.236,175.102,19.576,153.116
C08562=1087.492,91.241,-63.218,175.100,19.575,153.115
C08563=1087.486,90.991,-63.200,175.098,19.573,153.116
C08564=1087.480,90.742,-63.182,175.096,19.572,153.116
C08565=1087.474,90.492,-63.164,175.094,19.570,153.116
C08566=1087.468,90.243,-63.147,175.092,19.568,153.115
C08567=1087.463,89.994,-63.129,175.090,19.566,153.115
C08568=1087.457,89.745,-63.111,175.087,19.565,153.116
C08569=1087.451,89.496,-63.094,175.086,19.563,153.116
C08570=1087.445,89.246,-63.076,175.084,19.561,153.116
C08571=1087.440,88.997,-63.058,175.082,19.560,153.115
C08572=1087.434,88.748,-63.040,175.080,19.558,153.115
C08573=1087.428,88.498,-63.023,175.078,19.557,153.116
C08574=1087.422,88.249,-63.005,175.076,19.555,153.116
C08575=1087.417,88.000,-62.987,175.074,19.553,153.116
C08576=1087.411,87.750,-62.969,175.072,19.551,153.116
C08577=1087.405,87.501,-62.952,175.071,19.550,153.115
C08578=1087.400,87.252,-62.934,175.068,19.548,153.115
C08579=1087.394,87.002,-62.916,175.066,19.546,153.115
C08580=1087.388,86.753,-62.899,175.064,19.545,153.116
C08581=1087.383,86.504,-62.881,175.062,19.543,153.116
C08582=1087.376,86.255,-62.863,175.061,19.541,153.115
C08583=1087.371,86.005,-62.846,175.058,19.539,153.115
C08584=1087.366,85.756,-62.829,175.057,19.538,153.115
C08585=1087.360,85.507,-62.811,175.055,19.536,153.115
C08586=1087.354,85.257,-62.793,175.053,19.534,153.115
C08587=1087.349,85.008,-62.776,175.051,19.532,153.115
C08588=1087.343,84.759,-62.758,175.049,19.531,153.115
C08589=1087.337,84.509,-62.740,175.047,19.529,153.115
C08590=1087.332,84.260,-62.723,175.045,19.528,153.115
C08591=1087.326,84.011,-62.706,175.043,19.526,153.115
C08592=1087.321,83.762,-62.688,175.041,19.524,153.115
C08593=1087.315,83.512,-62.670,175.039,19.522,153.115
C08594=1087.309,83.263,-62.653,175.037,19.520,153.115
C08595=1087.303,83.013,-62.637,175.035,19.519,153.115
C08596=1087.298,82.764,-62.619,175.033,19.517,153.115
C08597=1087.291,82.515,-62.601,175.032,19.515,153.115
C08598=1087.286,82.266,-62.584,175.029,19.513,153.115
C08599=1087.281,82.016,-62.567,175.028,19.512,153.115
C08600=1087.275,81.767,-62.549,175.026,19.510,153.115
C08601=1087.270,81.518,-62.532,175.024,19.508,153.115
C08602=1087.264,81.268,-62.514,175.022,19.506,153.115
C08603=1087.258,81.018,-62.497,175.020,19.505,153.115
C08604=1087.253,80.769,-62.479,175.018,19.503,153.115
C08605=1087.247,80.520,-62.462,175.017,19.501,153.115
C08606=1087.242,80.271,-62.445,175.014,19.499,153.115
C08607=1087.235,80.021,-62.427,175.013,19.498,153.115
C08608=1087.230,79.743,-62.408,175.011,19.496,153.115
C08609=1087.223,79.466,-62.388,175.008,19.494,153.115
C08610=1087.217,79.188,-62.370,175.006,19.492,153.115
C08611=1087.211,78.910,-62.350,175.004,19.489,153.115
C08612=1087.205,78.661,-62.333,175.002,19.488,153.115
C08613=1087.199,78.412,-62.316,175.000,19.486,153.115
C08614=1087.194,78.162,-62.299,174.999,19.484,153.115
C08615=1087.188,77.912,-62.281,174.996,19.482,153.115
C08616=1087.182,77.663,-62.263,174.995,19.480,153.115
C08617=1087.176,77.414,-62.247,174.993,19.478,153.115
C08618=1087.171,77.165,-62.230,174.991,19.477,153.115
C08619=1087.166,76.915,-62.213,174.989,19.475,153.115
C08620=1087.159,76.667,-62.196,174.987,19.473,153.115
C08621=1087.154,76.416,-62.179,174.985,19.471,153.115
C08622=1087.148,76.167,-62.161,174.984,19.470,153.114
C08623=1087.142,75.918,-62.144,174.981,19.468,153.114
C08624=1087.137,75.669,-62.127,174.980,19.466,153.114
C08625=1087.131,75.420,-62.110,174.978,19.464,153.114
C08626=1087.126,75.170,-62.093,174.976,19.463,153.114
C08627=1087.119,74.921,-62.075,174.974,19.461,153.114
C08628=1087.114,74.671,-62.059,174.972,19.459,153.114
C08629=1087.108,74.422,-62.041,174.970,19.457,153.114
C08630=1087.102,74.173,-62.025,174.969,19.456,153.114
C08631=1087.097,73.924,-62.007,174.966,19.454,153.114
C08632=1087.092,73.674,-61.990,174.965,19.452,153.114
C08633=1087.086,73.425,-61.974,174.962,19.450,153.114
C08634=1087.080,73.176,-61.957,174.961,19.449,153.114
C08635=1087.074,72.925,-61.940,174.959,19.447,153.114
C08636=1087.068,72.676,-61.922,174.957,19.445,153.114
C08637=1087.063,72.427,-61.906,174.955,19.443,153.114
C08638=1087.057,72.178,-61.889,174.954,19.442,153.114
C08639=1087.051,71.928,-61.872,174.951,19.439,153.114
C08640=1087.046,71.679,-61.855,174.950,19.438,153.114
C08641=1087.040,71.430,-61.838,174.948,19.436,153.114
C08642=1087.035,71.180,-61.821,174.946,19.434,153.114
C08643=1087.029,70.931,-61.805,174.944,19.432,153.114
C08644=1087.023,70.682,-61.787,174.942,19.431,153.114
C08645=1087.018,70.432,-61.770,174.940,19.429,153.114
C08646=1087.011,70.183,-61.753,174.939,19.427,153.114
C08647=1087.006,69.933,-61.736,174.936,19.425,153.114
C08648=1087.000,69.684,-61.720,174.935,19.423,153.113
C08649=1086.995,69.434,-61.703,174.934,19.422,153.113
C08650=1086.989,69.185,-61.686,174.931,19.420,153.113
C08651=1086.983,68.936,-61.669,174.930,19.418,153.113
C08652=1086.977,68.686,-61.653,174.928,19.416,153.113
C08653=1086.972,68.437,-61.635,174.926,19.415,153.113
C08654=1086.966,68.188,-61.619,174.924,19.413,153.113
C08655=1086.961,67.938,-61.602,174.922,19.411,153.113
C08656=1086.955,67.689,-61.586,174.920,19.409,153.113
C08657=1086.949,67.440,-61.568,174.919,19.407,153.113
C08658=1086.943,67.191,-61.552,174.917,19.405,153.113
C08659=1086.938,66.941,-61.535,174.915,19.403,153.113
C08660=1086.932,66.692,-61.519,174.913,19.401,153.113
C08661=1086.927,66.443,-61.502,174.911,19.400,153.113
C08662=1086.921,66.193,-61.485,174.909,19.398,153.113
C08663=1086.915,65.944,-61.469,174.908,19.396,153.113
C08664=1086.910,65.694,-61.452,174.906,19.394,153.113
C08665=1086.904,65.445,-61.436,174.904,19.392,153.113
C08666=1086.898,65.196,-61.418,174.902,19.390,153.113
C08667=1086.892,64.947,-61.402,174.900,19.389,153.113
C08668=1086.887,64.697,-61.385,174.899,19.387,153.113
C08669=1086.881,64.448,-61.369,174.897,19.385,153.113
C08670=1086.874,64.197,-61.352,174.895,19.384,153.113
C08671=1086.869,63.948,-61.336,174.893,19.381,153.112
C08672=1086.862,63.671,-61.318,174.891,19.379,153.112
C08673=1086.856,63.393,-61.299,174.889,19.378,153.112
C08674=1086.849,63.115,-61.280,174.887,19.376,153.112
C08675=1086.843,62.837,-61.263,174.885,19.374,153.112
C08676=1086.837,62.587,-61.246,174.884,19.372,153.112
C08677=1086.831,62.339,-61.229,174.881,19.370,153.112
C08678=1086.826,62.089,-61.213,174.880,19.368,153.112
C08679=1086.820,61.840,-61.196,174.877,19.366,153.112
C08680=1086.814,61.590,-61.180,174.876,19.365,153.112
C08681=1086.808,61.341,-61.164,174.875,19.363,153.112
C08682=1086.803,61.091,-61.147,174.872,19.361,153.112
C08683=1086.797,60.842,-61.131,174.871,19.359,153.112
C08684=1086.791,60.593,-61.114,174.869,19.357,153.112
C08685=1086.785,60.343,-61.098,174.867,19.356,153.112
C08686=1086.779,60.094,-61.082,174.865,19.353,153.112
C08687=1086.774,59.844,-61.065,174.864,19.352,153.112
C08688=1086.768,59.595,-61.049,174.861,19.350,153.112
C08689=1086.762,59.346,-61.033,174.860,19.348,153.112
C08690=1086.756,59.096,-61.016,174.858,19.346,153.112
C08691=1086.750,58.847,-61.000,174.856,19.344,153.111
C08692=1086.745,58.597,-60.983,174.855,19.343,153.111
C08693=1086.739,58.348,-60.967,174.853,19.341,153.111
C08694=1086.733,58.099,-60.951,174.851,19.339,153.111
C08695=1086.727,57.849,-60.934,174.849,19.337,153.111
C08696=1086.721,57.599,-60.919,174.848,19.335,153.111
C08697=1086.715,57.350,-60.903,174.845,19.333,153.111
C08698=1086.710,57.100,-60.886,174.844,19.332,153.111
C08699=1086.704,56.851,-60.869,174.843,19.330,153.111
C08700=1086.698,56.602,-60.853,174.840,19.328,153.111
C08701=1086.693,56.353,-60.837,174.839,19.326,153.111
C08702=1086.687,56.104,-60.821,174.837,19.324,153.111
C08703=1086.681,55.854,-60.805,174.835,19.322,153.111
C08704=1086.675,55.605,-60.789,174.833,19.320,153.111
C08705=1086.670,55.355,-60.772,174.832,19.319,153.111
C08706=1086.664,55.105,-60.756,174.829,19.317,153.111
C08707=1086.658,54.856,-60.740,174.828,19.315,153.110
C08708=1086.652,54.607,-60.724,174.827,19.313,153.110
C08709=1086.646,54.357,-60.707,174.824,19.311,153.110
C08710=1086.641,54.108,-60.692,174.823,19.310,153.110
C08711=1086.635,53.859,-60.676,174.821,19.307,153.110
C08712=1086.629,53.609,-60.660,174.819,19.306,153.110
C08713=1086.624,53.360,-60.643,174.817,19.303,153.110
C08714=1086.618,53.110,-60.627,174.816,19.302,153.110
C08715=1086.613,52.860,-60.611,174.814,19.300,153.110
C08716=1086.607,52.611,-60.595,174.812,19.298,153.110
C08717=1086.601,52.362,-60.579,174.811,19.296,153.110
C08718=1086.595,52.113,-60.563,174.809,19.294,153.110
C08719=1086.590,51.863,-60.547,174.807,19.292,153.110
C08720=1086.584,51.614,-60.531,174.806,19.291,153.110
C08721=1086.578,51.364,-60.515,174.804,19.288,153.110
C08722=1086.573,51.115,-60.499,174.802,19.287,153.109
C08723=1086.567,50.866,-60.483,174.800,19.285,153.109
C08724=1086.562,50.616,-60.466,174.799,19.283,153.109
C08725=1086.556,50.367,-60.450,174.796,19.281,153.109
C08726=1086.550,50.117,-60.435,174.795,19.279,153.109
C08727=1086.545,49.868,-60.419,174.794,19.277,153.109
C08728=1086.539,49.619,-60.402,174.791,19.275,153.109
C08729=1086.533,49.369,-60.387,174.790,19.274,153.109
C08730=1086.527,49.119,-60.371,174.788,19.271,153.109
C08731=1086.522,48.870,-60.355,174.786,19.270,153.109
C08732=1086.516,48.621,-60.339,174.784,19.268,153.109
C08733=1086.510,48.371,-60.323,174.783,19.266,153.109
C08734=1086.504,48.121,-60.307,174.782,19.264,153.109
C08735=1086.499,47.873,-60.291,174.779,19.261,153.108
C08736=1086.493,47.594,-60.273,174.778,19.260,153.108
C08737=1086.486,47.316,-60.256,174.776,19.257,153.108
C08738=1086.480,47.038,-60.238,174.774,19.255,153.108
C08739=1086.474,46.760,-60.221,174.772,19.253,153.108
C08740=1086.468,46.511,-60.204,174.770,19.251,153.108
C08741=1086.463,46.261,-60.189,174.769,19.249,153.108
C08742=1086.457,46.012,-60.173,174.767,19.247,153.108
C08743=1086.452,45.762,-60.157,174.765,19.246,153.108
C08744=1086.446,45.513,-60.141,174.763,19.243,153.108
C08745=1086.440,45.263,-60.126,174.762,19.242,153.108
C08746=1086.435,45.014,-60.110,174.760,19.240,153.107
C08747=1086.429,44.764,-60.094,174.758,19.238,153.107
C08748=1086.423,44.515,-60.078,174.757,19.236,153.107
C08749=1086.418,44.265,-60.063,174.755,19.234,153.107
C08750=1086.412,44.016,-60.047,174.753,19.232,153.107
C08751=1086.406,43.766,-60.031,174.752,19.230,153.107
C08752=1086.401,43.517,-60.015,174.750,19.228,153.107
C08753=1086.395,43.268,-60.000,174.749,19.226,153.107
C08754=1086.389,43.018,-59.984,174.746,19.224,153.107
C08755=1086.384,42.769,-59.969,174.745,19.222,153.107
C08756=1086.378,42.519,-59.953,174.744,19.220,153.107
C08757=1086.372,42.270,-59.937,174.741,19.218,153.107
C08758=1086.366,42.020,-59.922,174.740,19.216,153.106
C08759=1086.360,41.772,-59.906,174.738,19.214,153.106
C08760=1086.355,41.522,-59.891,174.736,19.213,153.106
C08761=1086.349,41.272,-59.875,174.735,19.211,153.106
C08762=1086.344,41.023,-59.859,174.733,19.209,153.106
C08763=1086.337,40.773,-59.844,174.731,19.207,153.106
C08764=1086.332,40.523,-59.829,174.730,19.205,153.106
C08765=1086.326,40.275,-59.813,174.728,19.203,153.106
C08766=1086.321,40.025,-59.797,174.727,19.201,153.106
C08767=1086.315,39.775,-59.781,174.724,19.199,153.106
C08768=1086.309,39.526,-59.766,174.723,19.197,153.106
C08769=1086.303,39.276,-59.751,174.722,19.196,153.105
C08770=1086.298,39.026,-59.735,174.719,19.194,153.106
C08771=1086.292,38.778,-59.719,174.718,19.192,153.105
C08772=1086.286,38.528,-59.704,174.716,19.190,153.105
C08773=1086.280,38.278,-59.689,174.715,19.188,153.105
C08774=1086.275,38.030,-59.673,174.713,19.186,153.105
C08775=1086.269,37.780,-59.658,174.711,19.183,153.105
C08776=1086.263,37.530,-59.643,174.710,19.182,153.105
C08777=1086.258,37.281,-59.627,174.708,19.180,153.105
C08778=1086.252,37.031,-59.611,174.706,19.178,153.105
C08779=1086.245,36.782,-59.596,174.705,19.176,153.105
C08780=1086.240,36.532,-59.581,174.703,19.174,153.105
C08781=1086.234,36.283,-59.566,174.701,19.172,153.104
C08782=1086.229,36.034,-59.550,174.700,19.171,153.104
C08783=1086.223,35.784,-59.535,174.698,19.168,153.104
C08784=1086.217,35.534,-59.520,174.696,19.167,153.104
C08785=1086.212,35.285,-59.505,174.695,19.165,153.104
C08786=1086.205,35.036,-59.490,174.693,19.163,153.104
C08787=1086.199,34.786,-59.473,174.691,19.161,153.104
C08788=1086.194,34.537,-59.458,174.690,19.159,153.104
C08789=1086.188,34.287,-59.443,174.688,19.157,153.104
C08790=1086.183,34.038,-59.428,174.687,19.156,153.104
C08791=1086.176,33.788,-59.413,174.684,19.153,153.104
C08792=1086.171,33.538,-59.398,174.683,19.151,153.104
C08793=1086.165,33.289,-59.383,174.682,19.149,153.103
C08794=1086.159,33.040,-59.367,174.680,19.147,153.103
C08795=1086.154,32.791,-59.352,174.678,19.145,153.103
C08796=1086.148,32.541,-59.337,174.677,19.144,153.103
C08797=1086.142,32.291,-59.321,174.675,19.142,153.103
C08798=1086.136,32.042,-59.306,174.673,19.140,153.103
C08799=1086.131,31.792,-59.291,174.672,19.138,153.103
C08800=1086.124,31.514,-59.274,174.670,19.136,153.103
C08801=1086.118,31.236,-59.257,174.668,19.133,153.103
C08802=1086.111,30.958,-59.240,174.666,19.132,153.103
C08803=1086.105,30.680,-59.224,174.664,19.129,153.102
C08804=1086.100,30.431,-59.209,174.663,19.128,153.102
C08805=1086.093,30.181,-59.194,174.661,19.125,153.102
C08806=1086.088,29.932,-59.178,174.659,19.124,153.102
C08807=1086.082,29.682,-59.163,174.658,19.122,153.102
C08808=1086.077,29.433,-59.148,174.656,19.120,153.102
C08809=1086.070,29.183,-59.133,174.655,19.117,153.102
C08810=1086.065,28.934,-59.118,174.653,19.116,153.102
C08811=1086.059,28.684,-59.103,174.651,19.113,153.102
C08812=1086.054,28.435,-59.088,174.650,19.112,153.102
C08813=1086.047,28.185,-59.073,174.648,19.110,153.102
C08814=1086.042,27.936,-59.058,174.646,19.108,153.101
C08815=1086.036,27.686,-59.043,174.645,19.106,153.101
C08816=1086.030,27.437,-59.028,174.643,19.104,153.101
C08817=1086.025,27.187,-59.013,174.641,19.102,153.101
C08818=1086.019,26.938,-58.998,174.640,19.100,153.101
C08819=1086.013,26.688,-58.983,174.638,19.098,153.101
C08820=1086.007,26.439,-58.968,174.637,19.096,153.101
C08821=1086.001,26.190,-58.953,174.635,19.095,153.101
C08822=1085.995,25.940,-58.938,174.633,19.093,153.101
C08823=1085.990,25.691,-58.923,174.632,19.091,153.101
C08824=1085.983,25.441,-58.909,174.630,19.089,153.101
C08825=1085.978,25.191,-58.894,174.628,19.086,153.100
C08826=1085.972,24.942,-58.879,174.627,19.085,153.100
C08827=1085.966,24.693,-58.864,174.626,19.083,153.100
C08828=1085.961,24.443,-58.849,174.623,19.081,153.100
C08829=1085.955,24.194,-58.834,174.622,19.079,153.100
C08830=1085.948,23.944,-58.819,174.621,19.077,153.100
C08831=1085.944,23.694,-58.805,174.619,19.075,153.100
C08832=1085.938,23.445,-58.790,174.617,19.073,153.100
C08833=1085.932,23.196,-58.775,174.616,19.072,153.100
C08834=1085.927,22.946,-58.760,174.614,19.069,153.100
C08835=1085.920,22.697,-58.745,174.612,19.068,153.100
C08836=1085.915,22.447,-58.731,174.611,19.066,153.099
C08837=1085.908,22.197,-58.716,174.609,19.064,153.099
C08838=1085.903,21.948,-58.701,174.608,19.062,153.099
C08839=1085.897,21.699,-58.686,174.606,19.060,153.099
C08840=1085.891,21.450,-58.672,174.604,19.057,153.099
C08841=1085.886,21.199,-58.657,174.603,19.056,153.099
C08842=1085.880,20.950,-58.642,174.601,19.054,153.099
C08843=1085.874,20.701,-58.628,174.599,19.052,153.099
C08844=1085.868,20.451,-58.613,174.598,19.050,153.099
C08845=1085.863,20.202,-58.598,174.597,19.048,153.099
C08846=1085.857,19.952,-58.583,174.595,19.046,153.098
C08847=1085.851,19.703,-58.569,174.593,19.044,153.098
C08848=1085.845,19.453,-58.554,174.592,19.042,153.098
C08849=1085.839,19.204,-58.540,174.590,19.041,153.098
C08850=1085.834,18.954,-58.525,174.588,19.038,153.098
C08851=1085.828,18.704,-58.510,174.587,19.037,153.098
C08852=1085.822,18.455,-58.496,174.586,19.035,153.098
C08853=1085.816,18.206,-58.481,174.583,19.033,153.098
C08854=1085.810,17.956,-58.467,174.582,19.030,153.098
C08855=1085.804,17.707,-58.452,174.581,19.029,153.098
C08856=1085.799,17.457,-58.437,174.579,19.026,153.097
C08857=1085.793,17.207,-58.423,174.577,19.025,153.097
C08858=1085.787,16.958,-58.408,174.576,19.023,153.097
C08859=1085.781,16.708,-58.394,174.574,19.021,153.097
C08860=1085.776,16.459,-58.380,174.573,19.019,153.097
C08861=1085.769,16.210,-58.365,174.571,19.017,153.097
C08862=1085.765,15.960,-58.350,174.569,19.015,153.097
C08863=1085.759,15.711,-58.336,174.568,19.013,153.097
C08864=1085.752,15.434,-58.319,174.567,19.011,153.097
C08865=1085.746,15.157,-58.304,174.564,19.009,153.097
C08866=1085.739,14.881,-58.288,174.562,19.007,153.096
C08867=1085.733,14.604,-58.272,174.561,19.005,153.096
C08868=1085.727,14.355,-58.257,174.560,19.003,153.096
C08869=1085.721,14.105,-58.243,174.558,19.000,153.096
C08870=1085.715,13.856,-58.229,174.556,18.999,153.096
C08871=1085.709,13.605,-58.214,174.555,18.997,153.096
C08872=1085.703,13.356,-58.200,174.553,18.995,153.096
C08873=1085.698,13.107,-58.186,174.551,18.993,153.096
C08874=1085.691,12.857,-58.171,174.550,18.991,153.096
C08875=1085.686,12.608,-58.157,174.549,18.990,153.096
C08876=1085.680,12.359,-58.142,174.546,18.987,153.095
C08877=1085.674,12.108,-58.128,174.545,18.986,153.095
C08878=1085.668,11.859,-58.114,174.544,18.984,153.095
C08879=1085.662,11.609,-58.099,174.542,18.982,153.095
C08880=1085.656,11.360,-58.085,174.540,18.980,153.095
C08881=1085.651,11.111,-58.071,174.539,18.978,153.095
C08882=1085.645,10.860,-58.057,174.537,18.976,153.095
C08883=1085.639,10.611,-58.042,174.535,18.974,153.095
C08884=1085.633,10.362,-58.028,174.534,18.972,153.095
C08885=1085.627,10.112,-58.013,174.533,18.970,153.095
C08886=1085.622,9.863,-58.000,174.531,18.968,153.095
C08887=1085.615,9.614,-57.986,174.529,18.966,153.094
C08888=1085.609,9.364,-57.971,174.528,18.965,153.094
C08889=1085.603,9.114,-57.957,174.526,18.962,153.094
C08890=1085.598,8.865,-57.943,174.524,18.961,153.094
C08891=1085.592,8.615,-57.929,174.523,18.959,153.094
C08892=1085.586,8.365,-57.915,174.522,18.957,153.094
C08893=1085.580,8.116,-57.900,174.520,18.955,153.094
C08894=1085.575,7.867,-57.886,174.518,18.953,153.094
C08895=1085.569,7.616,-57.872,174.517,18.951,153.094
C08896=1085.563,7.367,-57.858,174.515,18.949,153.094
C08897=1085.557,7.118,-57.844,174.513,18.947,153.094
C08898=1085.551,6.868,-57.830,174.512,18.945,153.093
C08899=1085.545,6.619,-57.815,174.511,18.944,153.093
C08900=1085.539,6.369,-57.802,174.509,18.941,153.093
C08901=1085.534,6.120,-57.788,174.507,18.940,153.093
C08902=1085.528,5.870,-57.773,174.506,18.938,153.093
C08903=1085.522,5.621,-57.759,174.505,18.936,153.093
C08904=1085.516,5.371,-57.746,174.503,18.934,153.093
C08905=1085.510,5.122,-57.732,174.501,18.932,153.093
C08906=1085.504,4.872,-57.717,174.500,18.930,153.093
C08907=1085.499,4.622,-57.703,174.498,18.928,153.093
C08908=1085.493,4.373,-57.689,174.497,18.926,153.092
C08909=1085.488,4.123,-57.675,174.495,18.924,153.092
C08910=1085.482,3.874,-57.661,174.494,18.922,153.092
C08911=1085.475,3.624,-57.647,174.492,18.920,153.092
C08912=1085.470,3.375,-57.633,174.490,18.918,153.092
C08913=1085.464,3.125,-57.619,174.489,18.917,153.092
C08914=1085.459,2.876,-57.605,174.487,18.914,153.092
C08915=1085.453,2.626,-57.592,174.486,18.913,153.092
C08916=1085.447,2.376,-57.577,174.484,18.911,153.092
C08917=1085.441,2.127,-57.563,174.483,18.909,153.091
C08918=1085.435,1.878,-57.549,174.481,18.907,153.091
C08919=1085.430,1.628,-57.536,174.479,18.905,153.091
C08920=1085.424,1.378,-57.522,174.478,18.903,153.091
C08921=1085.418,1.128,-57.508,174.477,18.901,153.091
C08922=1085.412,0.879,-57.494,174.475,18.899,153.091
C08923=1085.406,0.630,-57.480,174.473,18.897,153.091
C08924=1085.401,0.380,-57.466,174.472,18.895,153.091
C08925=1085.395,0.131,-57.452,174.471,18.894,153.091
C08926=1085.390,-0.119,-57.438,174.469,18.891,153.091
C08927=1085.383,-0.368,-57.425,174.467,18.889,153.090
C08928=1085.377,-0.643,-57.410,174.466,18.888,153.090
C08929=1085.371,-0.918,-57.394,174.464,18.885,153.090
C08930=1085.365,-1.193,-57.379,174.463,18.883,153.090
C08931=1085.358,-1.467,-57.363,174.461,18.881,153.090
C08932=1085.353,-1.717,-57.349,174.459,18.879,153.090
C08933=1085.347,-1.966,-57.336,174.458,18.877,153.090
C08934=1085.341,-2.216,-57.322,174.456,18.875,153.090
C08935=1085.336,-2.465,-57.308,174.454,18.873,153.090
C08936=1085.330,-2.715,-57.295,174.453,18.871,153.089
C08937=1085.323,-2.965,-57.281,174.451,18.869,153.089
C08938=1085.318,-3.214,-57.267,174.450,18.867,153.089
C08939=1085.312,-3.464,-57.253,174.448,18.866,153.089
C08940=1085.306,-3.713,-57.240,174.447,18.864,153.089
C08941=1085.301,-3.963,-57.226,174.445,18.862,153.089
C08942=1085.294,-4.212,-57.213,174.444,18.860,153.089
C08943=1085.289,-4.462,-57.199,174.442,18.858,153.089
C08944=1085.283,-4.712,-57.185,174.441,18.856,153.089
C08945=1085.277,-4.961,-57.171,174.439,18.854,153.089
C08946=1085.271,-5.211,-57.158,174.438,18.852,153.088
C08947=1085.265,-5.460,-57.144,174.436,18.850,153.088
C08948=1085.259,-5.710,-57.130,174.435,18.849,153.088
C08949=1085.253,-5.959,-57.117,174.434,18.847,153.088
C08950=1085.248,-6.209,-57.104,174.431,18.845,153.088
C08951=1085.241,-6.459,-57.090,174.430,18.843,153.088
C08952=1085.236,-6.709,-57.077,174.429,18.841,153.088
C08953=1085.230,-6.958,-57.063,174.427,18.839,153.088
C08954=1085.224,-7.207,-57.049,174.425,18.837,153.088
C08955=1085.218,-7.457,-57.036,174.424,18.836,153.088
C08956=1085.212,-7.706,-57.022,174.423,18.833,153.088
C08957=1085.206,-7.955,-57.009,174.421,18.832,153.087
C08958=1085.201,-8.205,-56.995,174.419,18.829,153.087
C08959=1085.195,-8.455,-56.983,174.418,18.828,153.087
C08960=1085.189,-8.704,-56.969,174.416,18.826,153.087
C08961=1085.183,-8.954,-56.955,174.415,18.824,153.087
C08962=1085.177,-9.204,-56.941,174.413,18.822,153.087
C08963=1085.171,-9.453,-56.928,174.412,18.820,153.087
C08964=1085.165,-9.703,-56.914,174.410,18.819,153.087
C08965=1085.159,-9.953,-56.902,174.409,18.817,153.087
C08966=1085.154,-10.202,-56.888,174.407,18.815,153.087
C08967=1085.148,-10.452,-56.874,174.406,18.812,153.086
C08968=1085.142,-10.701,-56.861,174.404,18.811,153.086
C08969=1085.136,-10.951,-56.848,174.403,18.809,153.086
C08970=1085.131,-11.201,-56.834,174.401,18.807,153.086
C08971=1085.125,-11.450,-56.821,174.399,18.805,153.086
C08972=1085.118,-11.699,-56.808,174.398,18.803,153.086
C08973=1085.113,-11.949,-56.794,174.397,18.801,153.086
C08974=1085.107,-12.199,-56.781,174.395,18.800,153.086
C08975=1085.102,-12.448,-56.767,174.393,18.798,153.086
C08976=1085.095,-12.697,-56.754,174.392,18.796,153.086
C08977=1085.090,-12.948,-56.741,174.390,18.794,153.086
C08978=1085.084,-13.197,-56.728,174.389,18.792,153.085
C08979=1085.078,-13.446,-56.714,174.388,18.790,153.085
C08980=1085.072,-13.696,-56.700,174.386,18.788,153.085
C08981=1085.066,-13.946,-56.688,174.384,18.786,153.085
C08982=1085.061,-14.195,-56.674,174.383,18.784,153.085
C08983=1085.055,-14.444,-56.661,174.382,18.783,153.085
C08984=1085.050,-14.695,-56.648,174.380,18.780,153.085
C08985=1085.043,-14.944,-56.634,174.378,18.779,153.085
C08986=1085.037,-15.193,-56.621,174.377,18.777,153.085
C08987=1085.032,-15.443,-56.608,174.376,18.775,153.085
C08988=1085.026,-15.693,-56.595,174.374,18.774,153.085
C08989=1085.020,-15.943,-56.582,174.372,18.771,153.084
C08990=1085.014,-16.192,-56.569,174.371,18.769,153.084
C08991=1085.008,-16.441,-56.555,174.369,18.768,153.084
C08992=1085.001,-16.715,-56.540,174.367,18.765,153.084
C08993=1084.995,-16.987,-56.526,174.366,18.764,153.084
C08994=1084.989,-17.261,-56.512,174.365,18.762,153.084
C08995=1084.983,-17.534,-56.498,174.362,18.760,153.084
C08996=1084.976,-17.783,-56.485,174.361,18.758,153.084
C08997=1084.970,-18.033,-56.471,174.360,18.756,153.084
C08998=1084.964,-18.283,-56.459,174.359,18.754,153.084
C08999=1084.958,-18.532,-56.446,174.356,18.752,153.084
C09000=1084.953,-18.782,-56.432,174.355,18.751,153.084
C09001=1084.947,-19.031,-56.419,174.354,18.748,153.083
C09002=1084.941,-19.281,-56.407,174.352,18.747,153.083
C09003=1084.934,-19.530,-56.393,174.351,18.745,153.083
C09004=1084.929,-19.781,-56.380,174.349,18.743,153.083
C09005=1084.923,-20.030,-56.367,174.347,18.741,153.083
C09006=1084.917,-20.280,-56.354,174.346,18.739,153.083
C09007=1084.911,-20.529,-56.341,174.345,18.738,153.083
C09008=1084.905,-20.779,-56.329,174.343,18.736,153.083
C09009=1084.900,-21.028,-56.315,174.341,18.734,153.083
C09010=1084.894,-21.278,-56.303,174.340,18.732,153.083
C09011=1084.888,-21.527,-56.289,174.339,18.731,153.083
C09012=1084.882,-21.777,-56.277,174.337,18.728,153.082
C09013=1084.876,-22.026,-56.263,174.336,18.727,153.082
C09014=1084.871,-22.276,-56.250,174.334,18.724,153.082
C09015=1084.865,-22.525,-56.237,174.332,18.723,153.082
C09016=1084.859,-22.775,-56.224,174.331,18.721,153.082
C09017=1084.853,-23.025,-56.212,174.330,18.719,153.082
C09018=1084.847,-23.275,-56.199,174.328,18.718,153.082
C09019=1084.841,-23.524,-56.186,174.326,18.715,153.082
C09020=1084.836,-23.773,-56.173,174.325,18.714,153.082
C09021=1084.830,-24.023,-56.160,174.324,18.712,153.082
C09022=1084.824,-24.273,-56.147,174.322,18.710,153.082
C09023=1084.818,-24.522,-56.134,174.321,18.708,153.082
C09024=1084.812,-24.772,-56.122,174.319,18.707,153.081
C09025=1084.806,-25.021,-56.108,174.317,18.704,153.081
C09026=1084.800,-25.271,-56.096,174.316,18.703,153.081
C09027=1084.795,-25.522,-56.083,174.315,18.701,153.081
C09028=1084.789,-25.770,-56.070,174.313,18.699,153.081
C09029=1084.783,-26.020,-56.057,174.312,18.698,153.081
C09030=1084.777,-26.270,-56.045,174.310,18.695,153.081
C09031=1084.771,-26.519,-56.031,174.309,18.694,153.081
C09032=1084.765,-26.769,-56.019,174.307,18.692,153.081
C09033=1084.759,-27.019,-56.006,174.306,18.690,153.081
C09034=1084.754,-27.268,-55.994,174.304,18.688,153.081
C09035=1084.748,-27.517,-55.981,174.303,18.687,153.081
C09036=1084.742,-27.767,-55.968,174.301,18.684,153.080
C09037=1084.736,-28.017,-55.956,174.300,18.683,153.080
C09038=1084.729,-28.266,-55.942,174.298,18.681,153.080
C09039=1084.724,-28.516,-55.930,174.297,18.679,153.080
C09040=1084.718,-28.766,-55.917,174.296,18.678,153.080
C09041=1084.712,-29.016,-55.905,174.293,18.676,153.080
C09042=1084.706,-29.265,-55.892,174.292,18.674,153.080
C09043=1084.700,-29.514,-55.879,174.291,18.672,153.080
C09044=1084.694,-29.764,-55.867,174.289,18.671,153.080
C09045=1084.688,-30.014,-55.854,174.288,18.669,153.080
C09046=1084.682,-30.263,-55.841,174.287,18.667,153.080
C09047=1084.676,-30.513,-55.828,174.284,18.665,153.080
C09048=1084.670,-30.762,-55.817,174.283,18.663,153.080
C09049=1084.664,-31.012,-55.804,174.282,18.662,153.080
C09050=1084.658,-31.262,-55.792,174.280,18.660,153.079
C09051=1084.652,-31.511,-55.778,174.279,18.658,153.079
C09052=1084.646,-31.761,-55.766,174.277,18.657,153.079
C09053=1084.640,-32.011,-55.753,174.275,18.654,153.079
C09054=1084.635,-32.260,-55.741,174.274,18.653,153.079
C09055=1084.629,-32.510,-55.729,174.273,18.651,153.079
C09056=1084.622,-32.782,-55.715,174.271,18.649,153.079
C09057=1084.617,-33.054,-55.701,174.269,18.647,153.079
C09058=1084.610,-33.327,-55.687,174.268,18.645,153.079
C09059=1084.603,-33.599,-55.674,174.267,18.643,153.079
C09060=1084.598,-33.848,-55.662,174.265,18.642,153.079
C09061=1084.592,-34.098,-55.649,174.263,18.640,153.079
C09062=1084.586,-34.348,-55.636,174.262,18.638,153.079
C09063=1084.580,-34.598,-55.624,174.260,18.636,153.078
C09064=1084.575,-34.847,-55.612,174.259,18.635,153.078
C09065=1084.568,-35.097,-55.600,174.257,18.633,153.078
C09066=1084.562,-35.346,-55.586,174.256,18.631,153.078
C09067=1084.556,-35.596,-55.574,174.255,18.629,153.078
C09068=1084.550,-35.845,-55.562,174.253,18.627,153.078
C09069=1084.545,-36.095,-55.549,174.251,18.626,153.078
C09070=1084.539,-36.345,-55.537,174.250,18.624,153.078
C09071=1084.533,-36.595,-55.524,174.248,18.622,153.078
C09072=1084.527,-36.844,-55.512,174.247,18.621,153.078
C09073=1084.521,-37.093,-55.500,174.246,18.619,153.078
C09074=1084.515,-37.343,-55.487,174.244,18.617,153.078
C09075=1084.510,-37.592,-55.475,174.242,18.615,153.078
C09076=1084.504,-37.842,-55.463,174.241,18.614,153.078
C09077=1084.498,-38.092,-55.450,174.240,18.611,153.077
C09078=1084.492,-38.342,-55.438,174.238,18.610,153.077
C09079=1084.486,-38.591,-55.426,174.237,18.608,153.077
C09080=1084.480,-38.841,-55.413,174.235,18.607,153.077
C09081=1084.474,-39.091,-55.401,174.234,18.605,153.077
C09082=1084.469,-39.340,-55.389,174.232,18.603,153.077
C09083=1084.462,-39.590,-55.377,174.230,18.601,153.077
C09084=1084.456,-39.839,-55.364,174.229,18.600,153.077
C09085=1084.450,-40.089,-55.352,174.228,18.598,153.077
C09086=1084.444,-40.339,-55.341,174.226,18.597,153.077
C09087=1084.439,-40.589,-55.328,174.225,18.595,153.077
C09088=1084.433,-40.839,-55.316,174.224,18.593,153.077
C09089=1084.426,-41.088,-55.304,174.221,18.591,153.077
C09090=1084.421,-41.337,-55.291,174.220,18.589,153.077
C09091=1084.415,-41.587,-55.279,174.218,18.588,153.077
C09092=1084.408,-41.837,-55.267,174.217,18.586,153.077
C09093=1084.403,-42.086,-55.255,174.216,18.585,153.077
C09094=1084.396,-42.336,-55.243,174.214,18.583,153.077
C09095=1084.390,-42.585,-55.230,174.213,18.581,153.076
C09096=1084.385,-42.835,-55.219,174.212,18.580,153.076
C09097=1084.379,-43.085,-55.207,174.209,18.578,153.076
